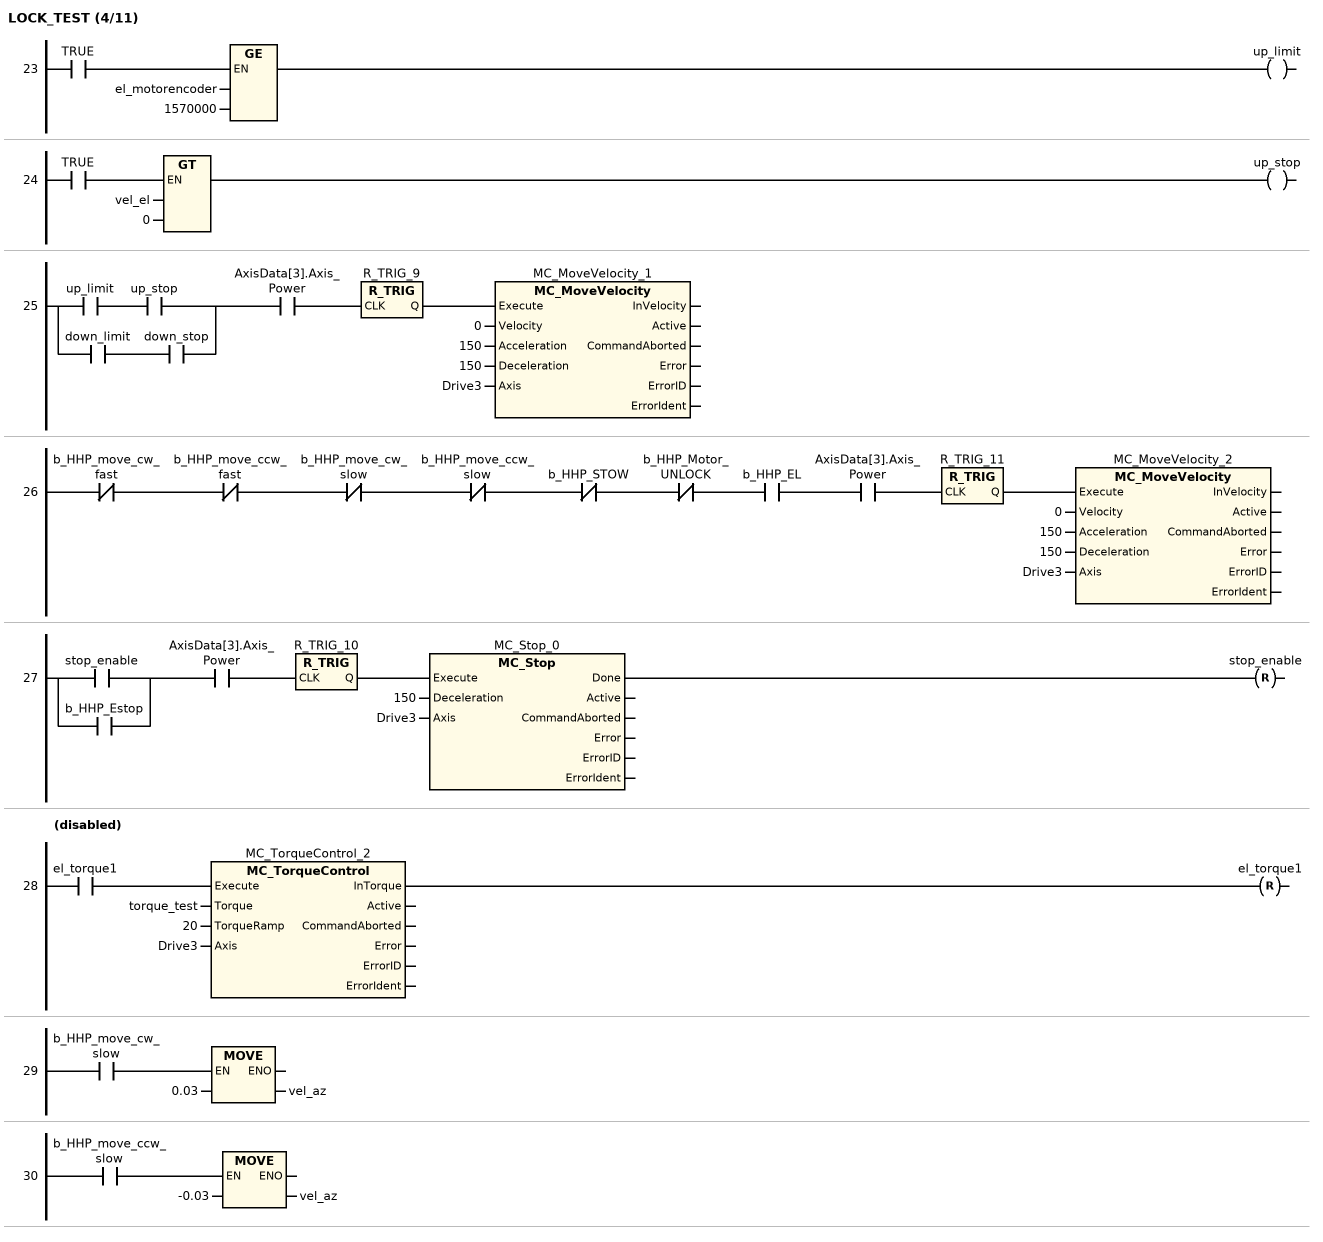
// NETWORK 23
up_limit := el_motorencoder >= 1570000;

// NETWORK 24
up_stop := vel_el > 0;

// NETWORK 25
R_TRIG_9(CLK := (up_limit AND up_stop OR down_limit AND down_stop) AND AxisData[3].Axis_Power); // R_TRIG
MC_MoveVelocity_1(
    Execute := R_TRIG_9.Q,
    Velocity := 0,
    Acceleration := 150,
    Deceleration := 150,
    Axis := Drive3); // MC_MoveVelocity

// NETWORK 26
R_TRIG_11(CLK := NOT b_HHP_move_cw_fast AND NOT b_HHP_move_ccw_fast AND NOT b_HHP_move_cw_slow AND NOT b_HHP_move_ccw_slow AND NOT b_HHP_STOW AND NOT b_HHP_Motor_UNLOCK AND b_HHP_EL AND AxisData[3].Axis_Power); // R_TRIG
MC_MoveVelocity_2(
    Execute := R_TRIG_11.Q,
    Velocity := 0,
    Acceleration := 150,
    Deceleration := 150,
    Axis := Drive3); // MC_MoveVelocity

// NETWORK 27
R_TRIG_10(CLK := (stop_enable OR b_HHP_Estop) AND AxisData[3].Axis_Power); // R_TRIG
MC_Stop_0(Execute := R_TRIG_10.Q, Deceleration := 150, Axis := Drive3); // MC_Stop
stop_enable R= MC_Stop_0.Done;

// NETWORK 28 (disabled)
// MC_TorqueControl_2(Execute := el_torque1, Torque := torque_test, TorqueRamp := 20, Axis := Drive3); // MC_TorqueControl
// el_torque1 R= MC_TorqueControl_2.InTorque;

// NETWORK 29
IF b_HHP_move_cw_slow THEN vel_az := 0.03; END_IF

// NETWORK 30
IF b_HHP_move_ccw_slow THEN vel_az := -0.03; END_IF

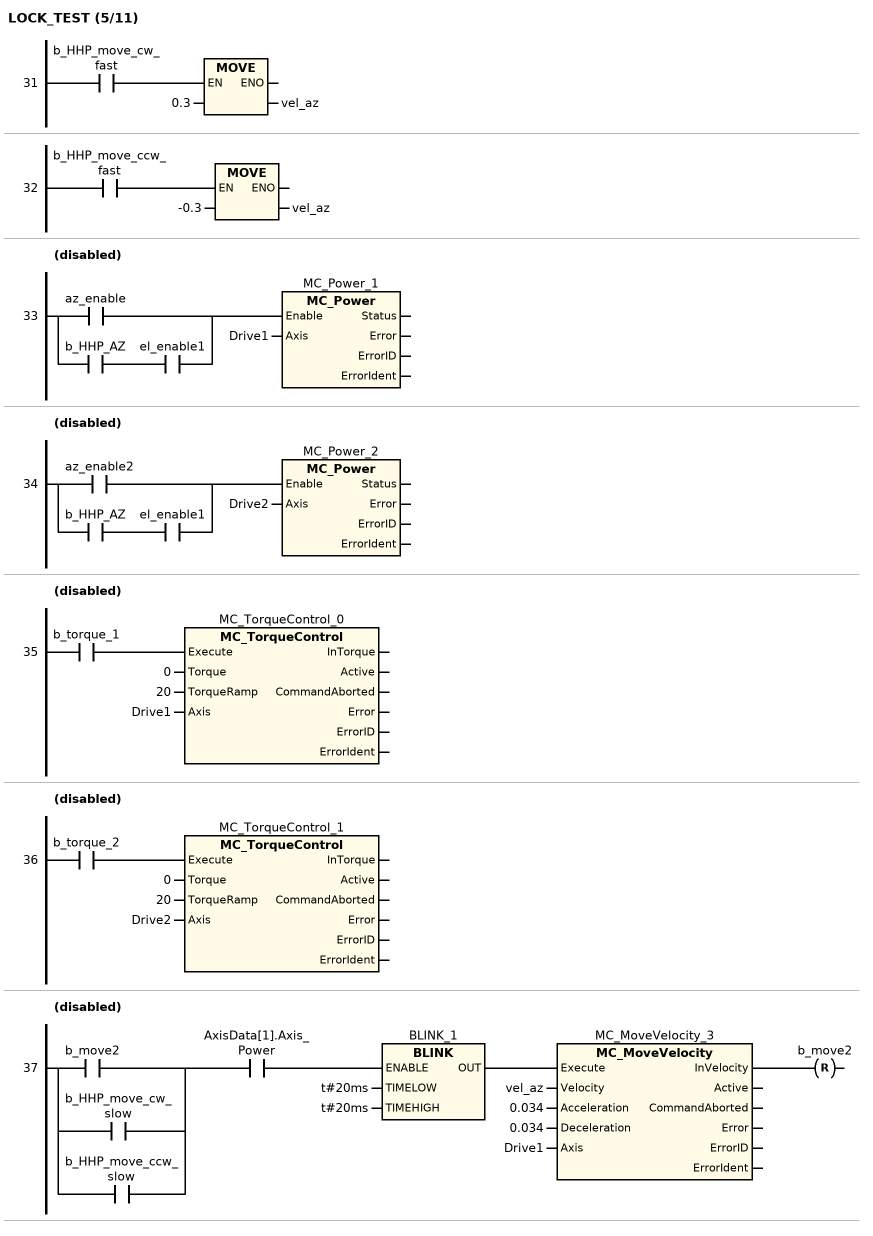
// NETWORK 31
IF b_HHP_move_cw_fast THEN vel_az := 0.3; END_IF

// NETWORK 32
IF b_HHP_move_ccw_fast THEN vel_az := -0.3; END_IF

// NETWORK 33 (disabled)
// MC_Power_1(Enable := az_enable OR b_HHP_AZ AND el_enable1, Axis := Drive1); // MC_Power

// NETWORK 34 (disabled)
// MC_Power_2(Enable := az_enable2 OR b_HHP_AZ AND el_enable1, Axis := Drive2); // MC_Power

// NETWORK 35 (disabled)
// MC_TorqueControl_0(Execute := b_torque_1, Torque := 0, TorqueRamp := 20, Axis := Drive1); // MC_TorqueControl

// NETWORK 36 (disabled)
// MC_TorqueControl_1(Execute := b_torque_2, Torque := 0, TorqueRamp := 20, Axis := Drive2); // MC_TorqueControl

// NETWORK 37 (disabled)
// BLINK_1(
//     ENABLE := (b_move2 OR b_HHP_move_cw_slow OR b_HHP_move_ccw_slow) AND AxisData[1].Axis_Power,
//     TIMELOW := t#20ms,
//     TIMEHIGH := t#20ms); // BLINK
// MC_MoveVelocity_3(
//     Execute := BLINK_1.OUT,
//     Velocity := vel_az,
//     Acceleration := 0.034,
//     Deceleration := 0.034,
//     Axis := Drive1); // MC_MoveVelocity
// b_move2 R= MC_MoveVelocity_3.InVelocity;

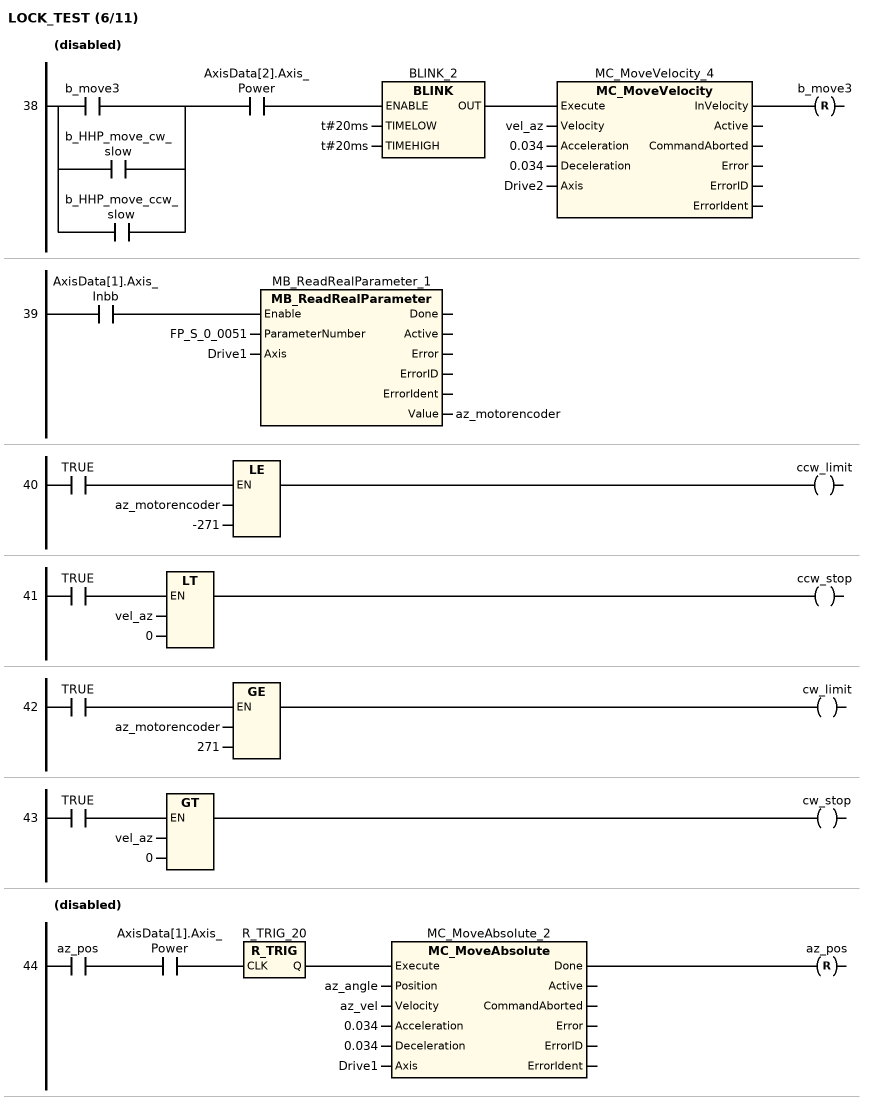
// NETWORK 38 (disabled)
// BLINK_2(
//     ENABLE := (b_move3 OR b_HHP_move_cw_slow OR b_HHP_move_ccw_slow) AND AxisData[2].Axis_Power,
//     TIMELOW := t#20ms,
//     TIMEHIGH := t#20ms); // BLINK
// MC_MoveVelocity_4(
//     Execute := BLINK_2.OUT,
//     Velocity := vel_az,
//     Acceleration := 0.034,
//     Deceleration := 0.034,
//     Axis := Drive2); // MC_MoveVelocity
// b_move3 R= MC_MoveVelocity_4.InVelocity;

// NETWORK 39
MB_ReadRealParameter_1(
    Enable := AxisData[1].Axis_Inbb,
    ParameterNumber := FP_S_0_0051,
    Axis := Drive1,
    Value => az_motorencoder); // MB_ReadRealParameter

// NETWORK 40
ccw_limit := az_motorencoder <= -271;

// NETWORK 41
ccw_stop := vel_az < 0;

// NETWORK 42
cw_limit := az_motorencoder >= 271;

// NETWORK 43
cw_stop := vel_az > 0;

// NETWORK 44 (disabled)
// R_TRIG_20(CLK := az_pos AND AxisData[1].Axis_Power); // R_TRIG
// MC_MoveAbsolute_2(
//     Execute := R_TRIG_20.Q,
//     Position := az_angle,
//     Velocity := az_vel,
//     Acceleration := 0.034,
//     Deceleration := 0.034,
//     Axis := Drive1); // MC_MoveAbsolute
// az_pos R= MC_MoveAbsolute_2.Done;

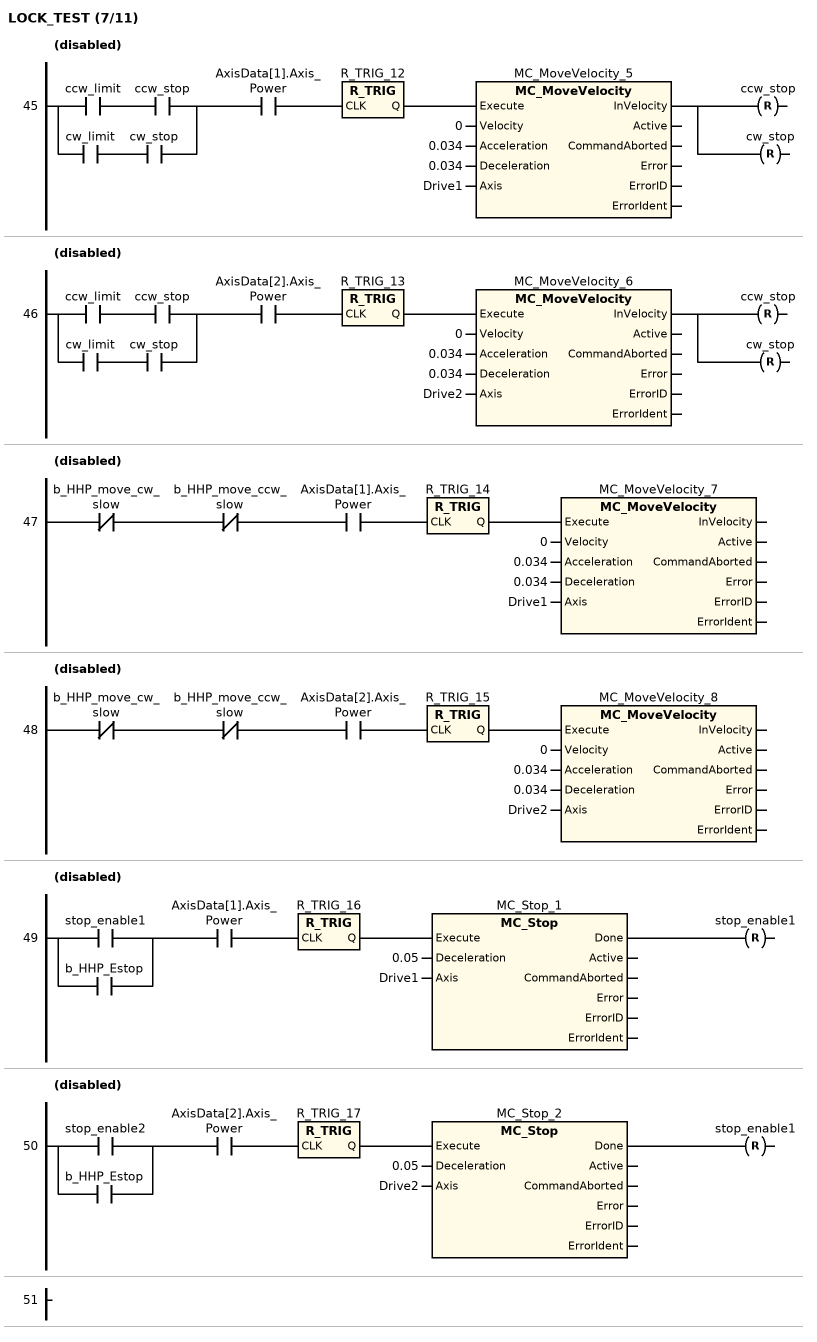
// NETWORK 45 (disabled)
// R_TRIG_12(CLK := (ccw_limit AND ccw_stop OR cw_limit AND cw_stop) AND AxisData[1].Axis_Power); // R_TRIG
// MC_MoveVelocity_5(
//     Execute := R_TRIG_12.Q,
//     Velocity := 0,
//     Acceleration := 0.034,
//     Deceleration := 0.034,
//     Axis := Drive1); // MC_MoveVelocity
// ccw_stop R= MC_MoveVelocity_5.InVelocity;
// cw_stop R= MC_MoveVelocity_5.InVelocity;

// NETWORK 46 (disabled)
// R_TRIG_13(CLK := (ccw_limit AND ccw_stop OR cw_limit AND cw_stop) AND AxisData[2].Axis_Power); // R_TRIG
// MC_MoveVelocity_6(
//     Execute := R_TRIG_13.Q,
//     Velocity := 0,
//     Acceleration := 0.034,
//     Deceleration := 0.034,
//     Axis := Drive2); // MC_MoveVelocity
// ccw_stop R= MC_MoveVelocity_6.InVelocity;
// cw_stop R= MC_MoveVelocity_6.InVelocity;

// NETWORK 47 (disabled)
// R_TRIG_14(CLK := NOT b_HHP_move_cw_slow AND NOT b_HHP_move_ccw_slow AND AxisData[1].Axis_Power); // R_TRIG
// MC_MoveVelocity_7(
//     Execute := R_TRIG_14.Q,
//     Velocity := 0,
//     Acceleration := 0.034,
//     Deceleration := 0.034,
//     Axis := Drive1); // MC_MoveVelocity

// NETWORK 48 (disabled)
// R_TRIG_15(CLK := NOT b_HHP_move_cw_slow AND NOT b_HHP_move_ccw_slow AND AxisData[2].Axis_Power); // R_TRIG
// MC_MoveVelocity_8(
//     Execute := R_TRIG_15.Q,
//     Velocity := 0,
//     Acceleration := 0.034,
//     Deceleration := 0.034,
//     Axis := Drive2); // MC_MoveVelocity

// NETWORK 49 (disabled)
// R_TRIG_16(CLK := (stop_enable1 OR b_HHP_Estop) AND AxisData[1].Axis_Power); // R_TRIG
// MC_Stop_1(Execute := R_TRIG_16.Q, Deceleration := 0.05, Axis := Drive1); // MC_Stop
// stop_enable1 R= MC_Stop_1.Done;

// NETWORK 50 (disabled)
// R_TRIG_17(CLK := (stop_enable2 OR b_HHP_Estop) AND AxisData[2].Axis_Power); // R_TRIG
// MC_Stop_2(Execute := R_TRIG_17.Q, Deceleration := 0.05, Axis := Drive2); // MC_Stop
// stop_enable1 R= MC_Stop_2.Done;

// NETWORK 51

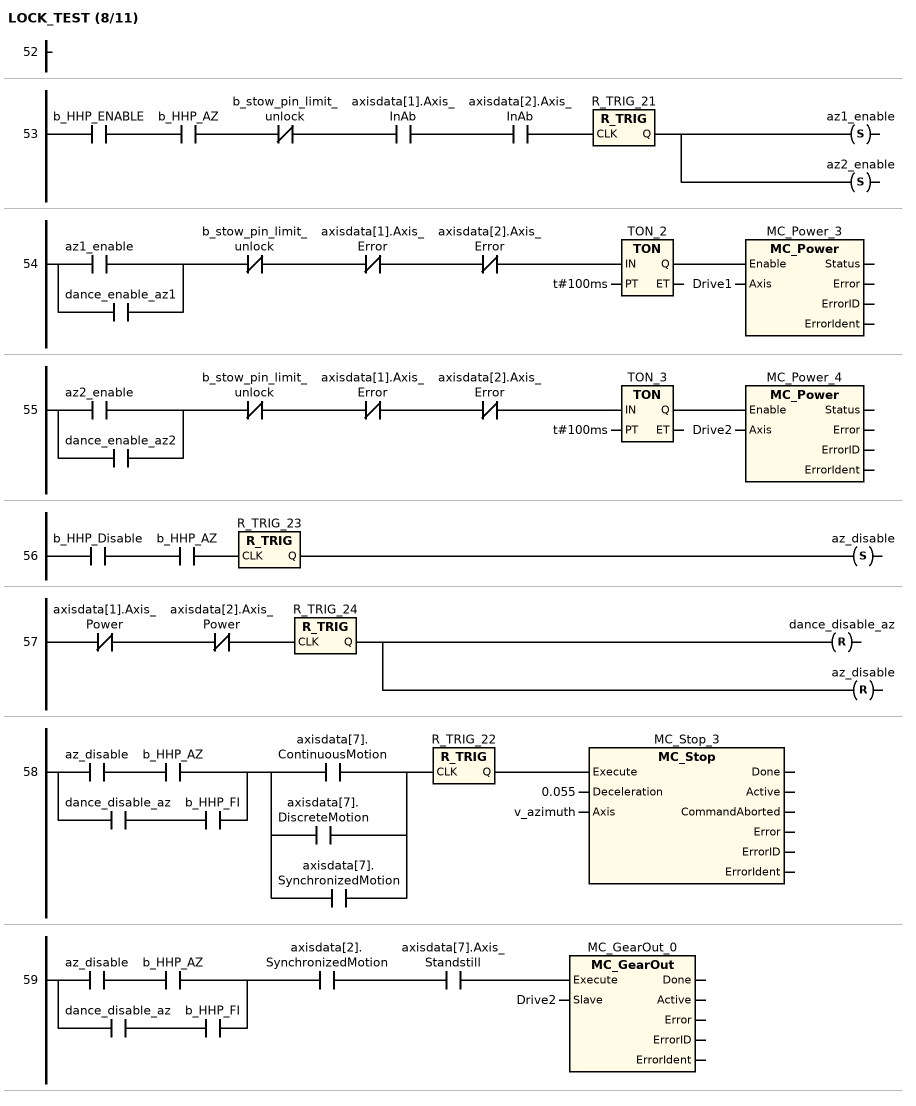
// NETWORK 52

// NETWORK 53
R_TRIG_21(CLK := b_HHP_ENABLE AND b_HHP_AZ AND NOT b_stow_pin_limit_unlock AND axisdata[1].Axis_InAb AND axisdata[2].Axis_InAb); // R_TRIG
az1_enable S= R_TRIG_21.Q;
az2_enable S= R_TRIG_21.Q;

// NETWORK 54
TON_2(IN := (az1_enable OR dance_enable_az1) AND NOT b_stow_pin_limit_unlock AND NOT axisdata[1].Axis_Error AND NOT axisdata[2].Axis_Error, PT := t#100ms); // TON
MC_Power_3(Enable := TON_2.Q, Axis := Drive1); // MC_Power

// NETWORK 55
TON_3(IN := (az2_enable OR dance_enable_az2) AND NOT b_stow_pin_limit_unlock AND NOT axisdata[1].Axis_Error AND NOT axisdata[2].Axis_Error, PT := t#100ms); // TON
MC_Power_4(Enable := TON_3.Q, Axis := Drive2); // MC_Power

// NETWORK 56
R_TRIG_23(CLK := b_HHP_Disable AND b_HHP_AZ); // R_TRIG
az_disable S= R_TRIG_23.Q;

// NETWORK 57
R_TRIG_24(CLK := NOT axisdata[1].Axis_Power AND NOT axisdata[2].Axis_Power); // R_TRIG
dance_disable_az R= R_TRIG_24.Q;
az_disable R= R_TRIG_24.Q;

// NETWORK 58
R_TRIG_22(CLK := (az_disable AND b_HHP_AZ OR dance_disable_az AND b_HHP_FI) AND (axisdata[7].ContinuousMotion OR axisdata[7].DiscreteMotion OR axisdata[7].SynchronizedMotion)); // R_TRIG
MC_Stop_3(Execute := R_TRIG_22.Q, Deceleration := 0.055, Axis := v_azimuth); // MC_Stop

// NETWORK 59
MC_GearOut_0(Execute := (az_disable AND b_HHP_AZ OR dance_disable_az AND b_HHP_FI) AND axisdata[2].SynchronizedMotion AND axisdata[7].Axis_Standstill, Slave := Drive2); // MC_GearOut

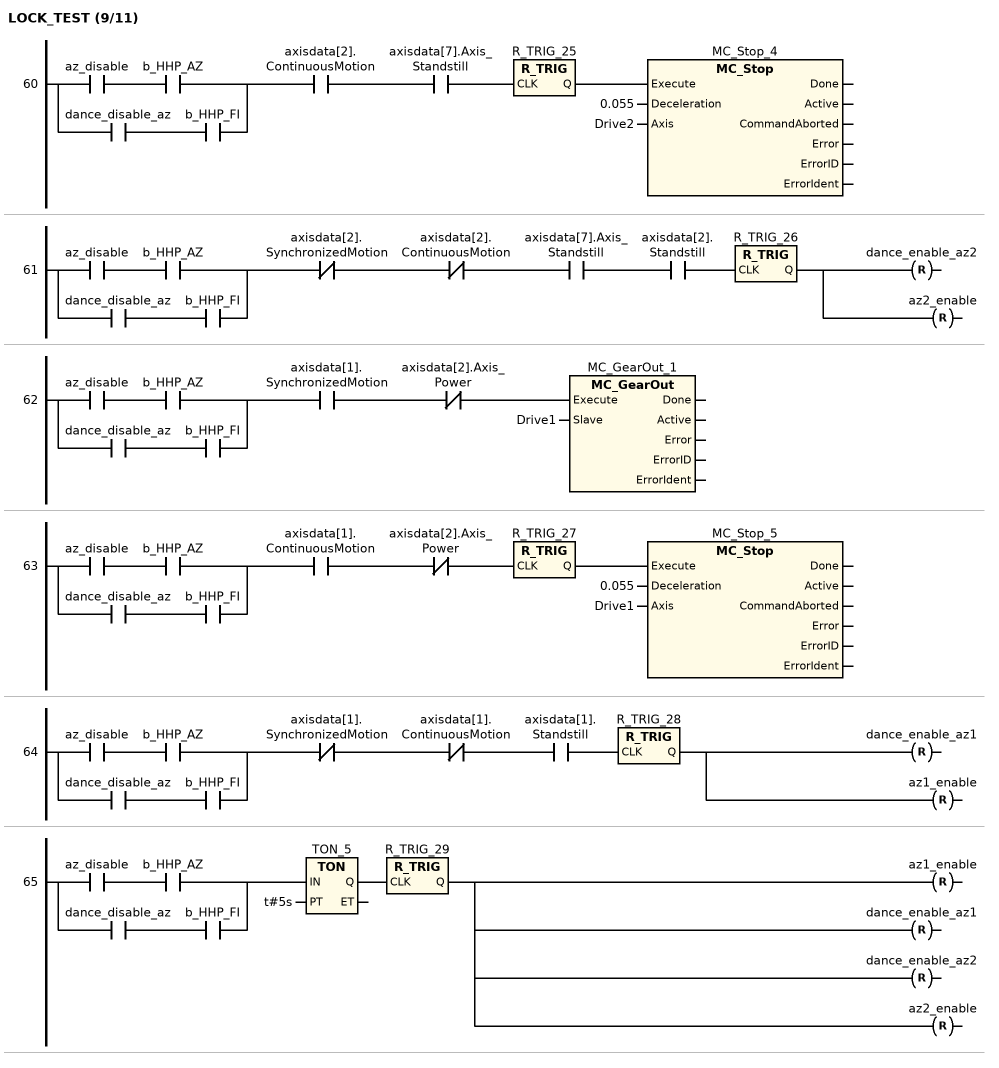
// NETWORK 60
R_TRIG_25(CLK := (az_disable AND b_HHP_AZ OR dance_disable_az AND b_HHP_FI) AND axisdata[2].ContinuousMotion AND axisdata[7].Axis_Standstill); // R_TRIG
MC_Stop_4(Execute := R_TRIG_25.Q, Deceleration := 0.055, Axis := Drive2); // MC_Stop

// NETWORK 61
R_TRIG_26(CLK := (az_disable AND b_HHP_AZ OR dance_disable_az AND b_HHP_FI) AND NOT axisdata[2].SynchronizedMotion AND NOT axisdata[2].ContinuousMotion AND axisdata[7].Axis_Standstill AND axisdata[2].Standstill); // R_TRIG
dance_enable_az2 R= R_TRIG_26.Q;
az2_enable R= R_TRIG_26.Q;

// NETWORK 62
MC_GearOut_1(Execute := (az_disable AND b_HHP_AZ OR dance_disable_az AND b_HHP_FI) AND axisdata[1].SynchronizedMotion AND NOT axisdata[2].Axis_Power, Slave := Drive1); // MC_GearOut

// NETWORK 63
R_TRIG_27(CLK := (az_disable AND b_HHP_AZ OR dance_disable_az AND b_HHP_FI) AND axisdata[1].ContinuousMotion AND NOT axisdata[2].Axis_Power); // R_TRIG
MC_Stop_5(Execute := R_TRIG_27.Q, Deceleration := 0.055, Axis := Drive1); // MC_Stop

// NETWORK 64
R_TRIG_28(CLK := (az_disable AND b_HHP_AZ OR dance_disable_az AND b_HHP_FI) AND NOT axisdata[1].SynchronizedMotion AND NOT axisdata[1].ContinuousMotion AND axisdata[1].Standstill); // R_TRIG
dance_enable_az1 R= R_TRIG_28.Q;
az1_enable R= R_TRIG_28.Q;

// NETWORK 65
TON_5(IN := az_disable AND b_HHP_AZ OR dance_disable_az AND b_HHP_FI, PT := t#5s); // TON
R_TRIG_29(CLK := TON_5.Q); // R_TRIG
az1_enable R= R_TRIG_29.Q;
dance_enable_az1 R= R_TRIG_29.Q;
dance_enable_az2 R= R_TRIG_29.Q;
az2_enable R= R_TRIG_29.Q;

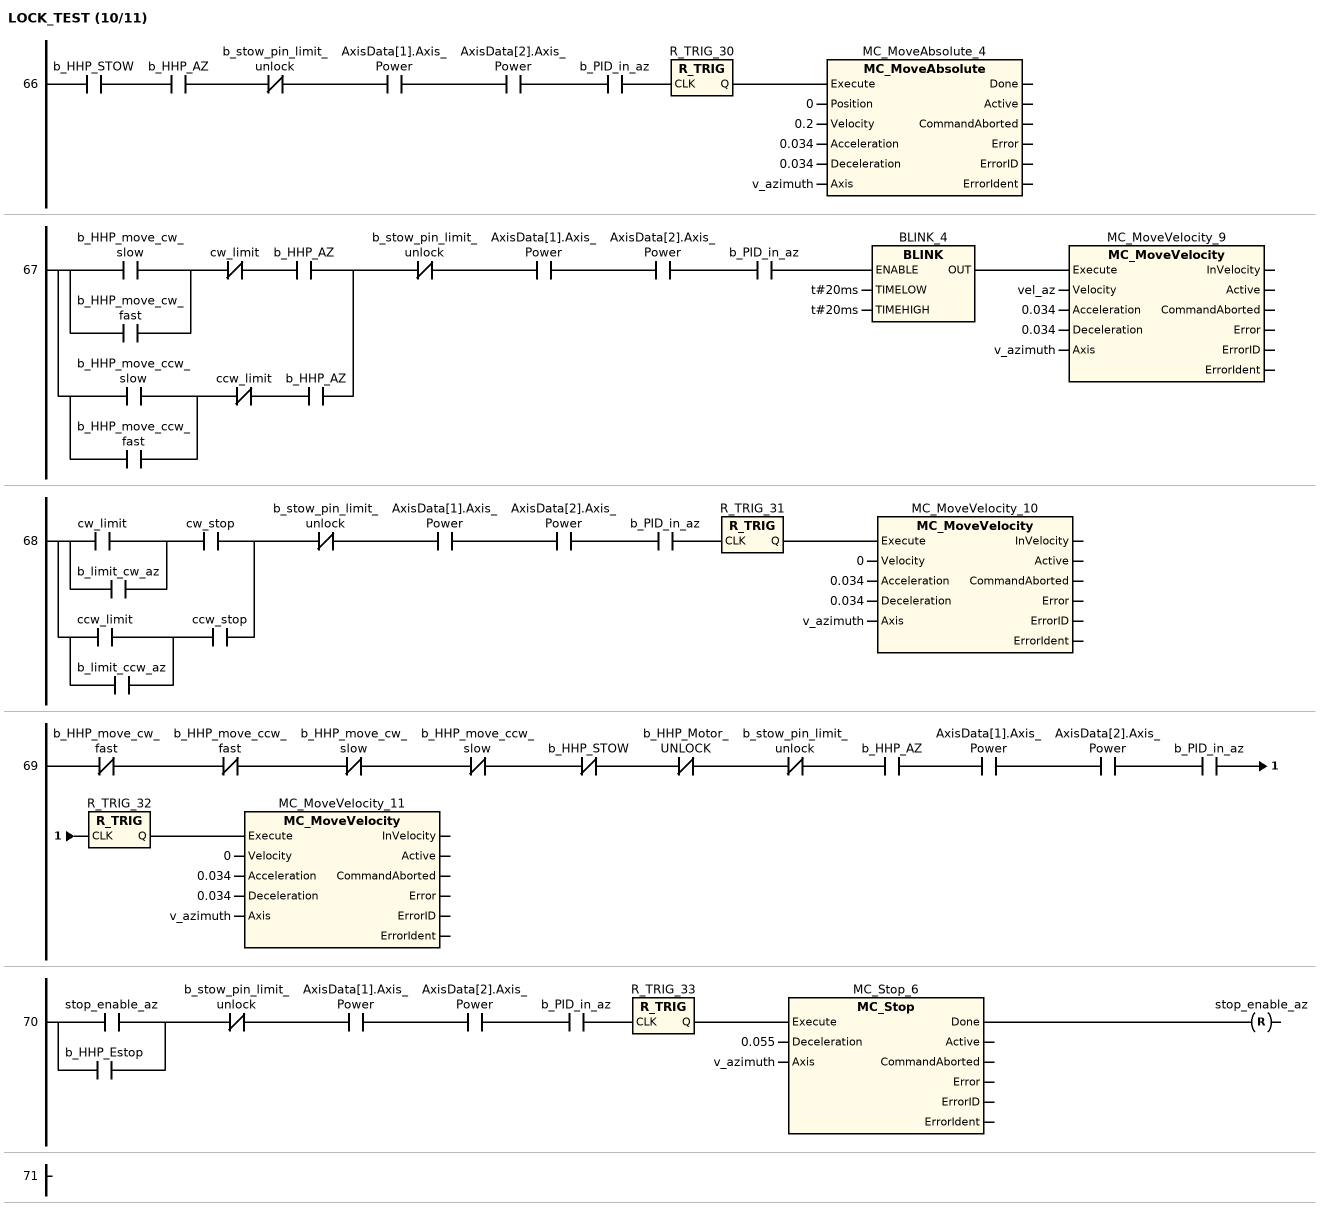
// NETWORK 66
R_TRIG_30(CLK := b_HHP_STOW AND b_HHP_AZ AND NOT b_stow_pin_limit_unlock AND AxisData[1].Axis_Power AND AxisData[2].Axis_Power AND b_PID_in_az); // R_TRIG
MC_MoveAbsolute_4(
    Execute := R_TRIG_30.Q,
    Position := 0,
    Velocity := 0.2,
    Acceleration := 0.034,
    Deceleration := 0.034,
    Axis := v_azimuth); // MC_MoveAbsolute

// NETWORK 67
BLINK_4(
    ENABLE := ((b_HHP_move_cw_slow OR b_HHP_move_cw_fast) AND NOT cw_limit AND b_HHP_AZ OR (b_HHP_move_ccw_slow OR b_HHP_move_ccw_fast) AND NOT ccw_limit AND b_HHP_AZ) AND NOT b_stow_pin_limit_unlock AND AxisData[1].Axis_Power AND AxisData[2].Axis_Power AND b_PID_in_az,
    TIMELOW := t#20ms,
    TIMEHIGH := t#20ms); // BLINK
MC_MoveVelocity_9(
    Execute := BLINK_4.OUT,
    Velocity := vel_az,
    Acceleration := 0.034,
    Deceleration := 0.034,
    Axis := v_azimuth); // MC_MoveVelocity

// NETWORK 68
R_TRIG_31(CLK := ((cw_limit OR b_limit_cw_az) AND cw_stop OR (ccw_limit OR b_limit_ccw_az) AND ccw_stop) AND NOT b_stow_pin_limit_unlock AND AxisData[1].Axis_Power AND AxisData[2].Axis_Power AND b_PID_in_az); // R_TRIG
MC_MoveVelocity_10(
    Execute := R_TRIG_31.Q,
    Velocity := 0,
    Acceleration := 0.034,
    Deceleration := 0.034,
    Axis := v_azimuth); // MC_MoveVelocity

// NETWORK 69
R_TRIG_32(CLK := NOT b_HHP_move_cw_fast AND NOT b_HHP_move_ccw_fast AND NOT b_HHP_move_cw_slow AND NOT b_HHP_move_ccw_slow AND NOT b_HHP_STOW AND NOT b_HHP_Motor_UNLOCK AND NOT b_stow_pin_limit_unlock AND b_HHP_AZ AND AxisData[1].Axis_Power AND AxisData[2].Axis_Power AND b_PID_in_az); // R_TRIG
MC_MoveVelocity_11(
    Execute := R_TRIG_32.Q,
    Velocity := 0,
    Acceleration := 0.034,
    Deceleration := 0.034,
    Axis := v_azimuth); // MC_MoveVelocity

// NETWORK 70
R_TRIG_33(CLK := (stop_enable_az OR b_HHP_Estop) AND NOT b_stow_pin_limit_unlock AND AxisData[1].Axis_Power AND AxisData[2].Axis_Power AND b_PID_in_az); // R_TRIG
MC_Stop_6(Execute := R_TRIG_33.Q, Deceleration := 0.055, Axis := v_azimuth); // MC_Stop
stop_enable_az R= MC_Stop_6.Done;

// NETWORK 71

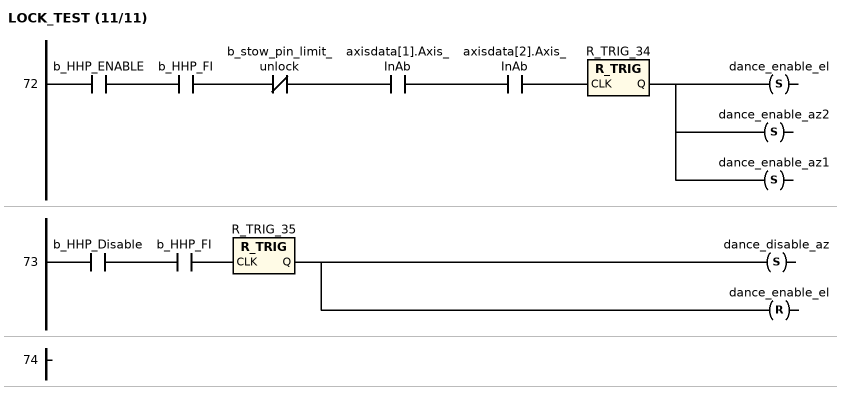
// NETWORK 72
R_TRIG_34(CLK := b_HHP_ENABLE AND b_HHP_FI AND NOT b_stow_pin_limit_unlock AND axisdata[1].Axis_InAb AND axisdata[2].Axis_InAb); // R_TRIG
dance_enable_el S= R_TRIG_34.Q;
dance_enable_az2 S= R_TRIG_34.Q;
dance_enable_az1 S= R_TRIG_34.Q;

// NETWORK 73
R_TRIG_35(CLK := b_HHP_Disable AND b_HHP_FI); // R_TRIG
dance_disable_az S= R_TRIG_35.Q;
dance_enable_el R= R_TRIG_35.Q;

// NETWORK 74

END_PROGRAM

// IndraMotionMlc1/Application/POUs/Motion/P_power_on_Sim
(*the program is built for power on the 3 axis under the contol of remote or local.
the elevation axis is the similar with the azimuth*)
PROGRAM P_power_on_Sim
VAR
(*<<<<<<<<definition of r_trig for detecting a rising edge>>>>>>>>>>>>>>*)
	fb_rtrig_p1: R_TRIG;
	fb_rtrig_p3: R_TRIG;
	fb_rtrig_p5: R_TRIG;
	fb_rtrig_az: R_TRIG;
	fb_rtrig_el: R_TRIG;
	fb_rtrig_FI: R_TRIG;
	fb_rtrig_en_remote: R_TRIG;
	fb_rtrig_en_TCP: R_TRIG;
(*<<<<<<<The function block Timer On Delay implements a turn-on delay>>>>>>*)
	ton_en_1: TON;
	ton_en_2: TON;
	ton_en_3: TON;
	ton_en_4: TON;
	ton_en_5: TON;
	ton_en_6: TON;
(*MC_Power function block controls the power connection (power on or off)*)
	FB_1_power: MC_Power;
	FB_2_power: MC_Power;
	FB_3_power: MC_Power;
	FB_4_power: MC_Power;
	FB_5_power: MC_Power;
	FB_6_power: MC_Power;
	b_1_enable_on: BOOL;
	b_2_enable_on: BOOL;
	b_3_enable_on: BOOL;
	b_4_enable_on: BOOL;
	b_5_enable_on: BOOL;
	b_6_enable_on: BOOL;
(*With "MB_GearInPos",it is possible to realize a motion of the slave axis which is phase synchronous to the master axis*)
	fb_gearinPos_1: MB_GearInPos;
	fb_gearin_2: MB_GearInPos;
	fb_gearinPos_3: MB_GearInPos;
	fb_gearin_4: MB_GearInPos;
	fb_gearinPos_5: MB_GearInPos;
	fb_gearin_6: MB_GearInPos;
	b_gearin_1_done: BOOL;
	
	b_gearin_5_done:BOOL;
(*"MC_MoveAbsolute" is used to move the drive to a preset absolute position.*)
	FB_move_master_az: MC_MoveAbsolute;
	FB_move_master_el: MC_MoveAbsolute;
	FB_move_master_FI: MC_MoveAbsolute;
	b_M_az_done: BOOL;
	b_M_el_done: BOOL;
	b_M_FI_done: BOOL;
(*MB_Home function block controls axes with incremental encoder when executing the "search home" sequence*)
	fb_home_az2: MB_Home;
	fb_home_el2: MB_Home;
	fb_home_FI2: MB_Home;
	b_home_az2_done: BOOL;
	b_home_el2_done: BOOL;
	b_home_FI2_done: BOOL;
(*<<<<<<<<<<<<<<<<<<<<<<<<<<<<<clear error>>>>>>>>>>>>>>>>>>>>>>>>>>>>>>>>>*)
	TCP_clear_error: BOOL;
	FB_clear_error_TCP: MB_WriteParameter;
	TCP_clear_done: BOOL;
(*add 2011 06 09 to delete 1sec delay*)
	fb_gearinPos_el: MB_GearInPos;
	b_gearin_el_done: BOOL;
	fb_gearout_el: MC_GearOut;
	rtrig_set_gearin_3: R_TRIG;
	b_gearin_3: BOOL;
	rtrig_reset_gearin_3: F_TRIG;
	ton_clear_on: TON;
	fb_gearinPos_FI: MB_GearInPos;
	test_111: BOOL;
	ssss: BOOL;
	test1: BOOL;
	test2: BOOL;
	test3: BOOL;
	TON_enable_az: ton;
	TON_enable_az2: ton;
	fb_gearPos_2: MB_GearInPos;
	TON_enable_el: ton;
	b_M_el_done_1: BOOL;
	R_TRIG_0: R_TRIG;
END_VAR

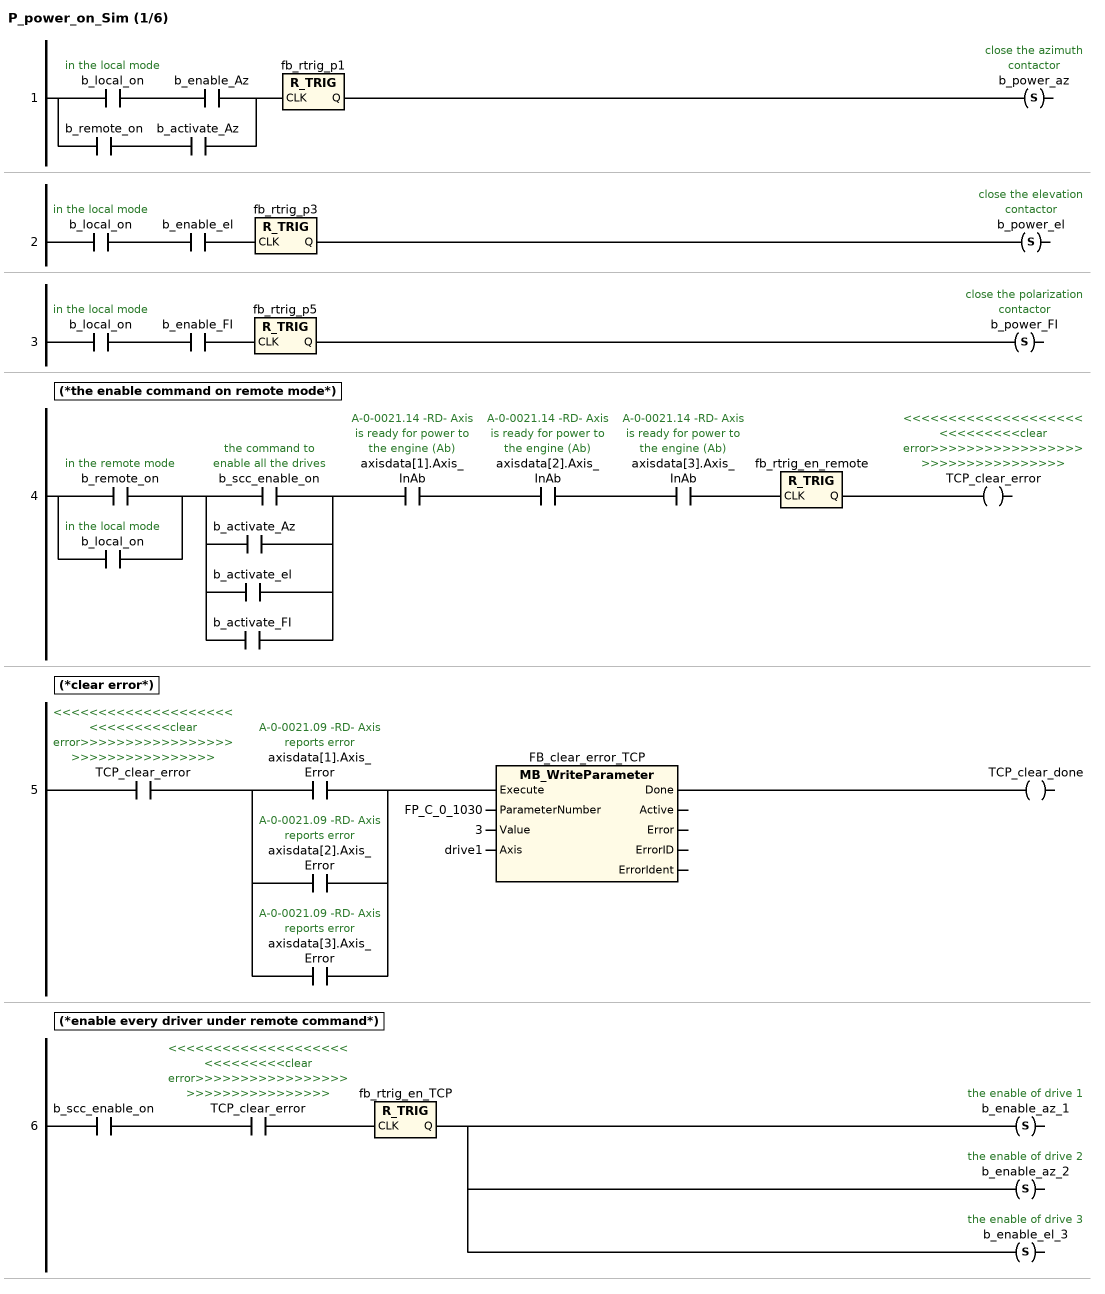
// NETWORK 1
//   fb_rtrig_p1: <<<<<<<<definition of r_trig for detecting a rising edge>>>>>>>>>>>>>>
//   b_local_on: in the local mode
//   b_power_az: close the azimuth contactor
fb_rtrig_p1(CLK := b_local_on AND b_enable_Az OR b_remote_on AND b_activate_Az); // R_TRIG
b_power_az S= fb_rtrig_p1.Q;

// NETWORK 2
//   b_local_on: in the local mode
//   b_power_el: close the elevation contactor
fb_rtrig_p3(CLK := b_local_on AND b_enable_el); // R_TRIG
b_power_el S= fb_rtrig_p3.Q;

// NETWORK 3
//   b_local_on: in the local mode
//   b_power_FI: close the polarization contactor
fb_rtrig_p5(CLK := b_local_on AND b_enable_FI); // R_TRIG
b_power_FI S= fb_rtrig_p5.Q;

// NETWORK 4
//   b_remote_on: in the remote mode
//   b_local_on: in the local mode
//   b_scc_enable_on: the command to enable all the drives
//   axisdata[1].Axis_InAb: A-0-0021.14 -RD- Axis is ready for power to the engine (Ab)
//   axisdata[2].Axis_InAb: A-0-0021.14 -RD- Axis is ready for power to the engine (Ab)
//   axisdata[3].Axis_InAb: A-0-0021.14 -RD- Axis is ready for power to the engine (Ab)
//   TCP_clear_error: <<<<<<<<<<<<<<<<<<<<<<<<<<<<<clear error>>>>>>>>>>>>>>>>>>>>>>>>>>>>>>>>>
// label: (*the enable command on remote mode*)
fb_rtrig_en_remote(CLK := (b_remote_on OR b_local_on) AND (b_scc_enable_on OR b_activate_Az OR b_activate_el OR b_activate_FI) AND axisdata[1].Axis_InAb AND axisdata[2].Axis_InAb AND axisdata[3].Axis_InAb); // R_TRIG
TCP_clear_error := fb_rtrig_en_remote.Q;

// NETWORK 5
//   TCP_clear_error: <<<<<<<<<<<<<<<<<<<<<<<<<<<<<clear error>>>>>>>>>>>>>>>>>>>>>>>>>>>>>>>>>
//   axisdata[1].Axis_Error: A-0-0021.09 -RD- Axis reports error
//   axisdata[2].Axis_Error: A-0-0021.09 -RD- Axis reports error
//   axisdata[3].Axis_Error: A-0-0021.09 -RD- Axis reports error
//   FP_C_0_1030: Command: Clear all control errors
//   drive1: Real axis "Drive1" with axis number 1
// label: (*clear error*)
FB_clear_error_TCP(
    Execute := TCP_clear_error AND (axisdata[1].Axis_Error OR axisdata[2].Axis_Error OR axisdata[3].Axis_Error),
    ParameterNumber := FP_C_0_1030,
    Value := 3,
    Axis := drive1); // MB_WriteParameter
TCP_clear_done := FB_clear_error_TCP.Done;

// NETWORK 6
//   TCP_clear_error: <<<<<<<<<<<<<<<<<<<<<<<<<<<<<clear error>>>>>>>>>>>>>>>>>>>>>>>>>>>>>>>>>
//   b_enable_az_1: the enable of drive 1
//   b_enable_az_2: the enable of drive 2
//   b_enable_el_3: the enable of drive 3
// label: (*enable every driver under remote command*)
fb_rtrig_en_TCP(CLK := b_scc_enable_on AND TCP_clear_error); // R_TRIG
b_enable_az_1 S= fb_rtrig_en_TCP.Q;
b_enable_az_2 S= fb_rtrig_en_TCP.Q;
b_enable_el_3 S= fb_rtrig_en_TCP.Q;

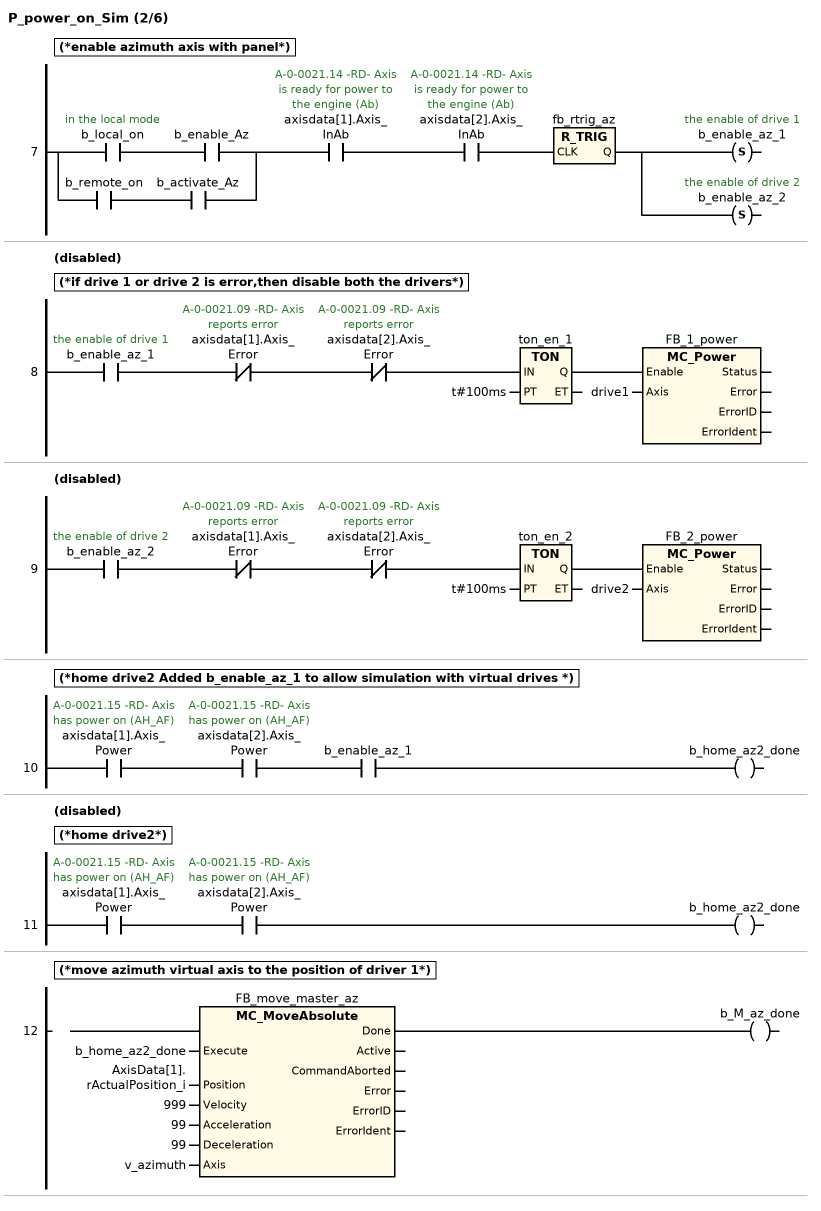
// NETWORK 7
//   b_local_on: in the local mode
//   axisdata[1].Axis_InAb: A-0-0021.14 -RD- Axis is ready for power to the engine (Ab)
//   axisdata[2].Axis_InAb: A-0-0021.14 -RD- Axis is ready for power to the engine (Ab)
//   b_enable_az_1: the enable of drive 1
//   b_enable_az_2: the enable of drive 2
// label: (*enable azimuth axis with panel*)
fb_rtrig_az(CLK := (b_local_on AND b_enable_Az OR b_remote_on AND b_activate_Az) AND axisdata[1].Axis_InAb AND axisdata[2].Axis_InAb); // R_TRIG
b_enable_az_1 S= fb_rtrig_az.Q;
b_enable_az_2 S= fb_rtrig_az.Q;

// NETWORK 8 (disabled)
//   FB_1_power: MC_Power function block controls the power connection (power on or off)
//   ton_en_1: <<<<<<<The function block Timer On Delay implements a turn-on delay>>>>>>
//   b_enable_az_1: the enable of drive 1
//   axisdata[1].Axis_Error: A-0-0021.09 -RD- Axis reports error
//   axisdata[2].Axis_Error: A-0-0021.09 -RD- Axis reports error
//   drive1: Real axis "Drive1" with axis number 1
// label: (*if drive 1 or drive 2 is error,then disable both the drivers*)
// ton_en_1(IN := b_enable_az_1 AND NOT axisdata[1].Axis_Error AND NOT axisdata[2].Axis_Error, PT := t#100ms); // TON
// FB_1_power(Enable := ton_en_1.Q, Axis := drive1); // MC_Power

// NETWORK 9 (disabled)
//   b_enable_az_2: the enable of drive 2
//   axisdata[1].Axis_Error: A-0-0021.09 -RD- Axis reports error
//   axisdata[2].Axis_Error: A-0-0021.09 -RD- Axis reports error
//   drive2: Real axis "Drive2" with axis number 2
// ton_en_2(IN := b_enable_az_2 AND NOT axisdata[1].Axis_Error AND NOT axisdata[2].Axis_Error, PT := t#100ms); // TON
// FB_2_power(Enable := ton_en_2.Q, Axis := drive2); // MC_Power

// NETWORK 10
//   axisdata[1].Axis_Power: A-0-0021.15 -RD- Axis has power on (AH_AF)
//   axisdata[2].Axis_Power: A-0-0021.15 -RD- Axis has power on (AH_AF)
// label: (*home drive2 Added b_enable_az_1 to allow simulation with virtual drives *)
b_home_az2_done := axisdata[1].Axis_Power AND axisdata[2].Axis_Power AND b_enable_az_1;

// NETWORK 11 (disabled)
//   axisdata[1].Axis_Power: A-0-0021.15 -RD- Axis has power on (AH_AF)
//   axisdata[2].Axis_Power: A-0-0021.15 -RD- Axis has power on (AH_AF)
// label: (*home drive2*)
// b_home_az2_done := axisdata[1].Axis_Power AND axisdata[2].Axis_Power;

// NETWORK 12
//   FB_move_master_az: "MC_MoveAbsolute" is used to move the drive to a preset absolute position.
//   AxisData[1].rActualPosition_i: A-0-0100 -RD- Actual position
//   v_azimuth: Virtual axis "v_azimuth" with axis number 7
// label: (*move azimuth virtual axis to the position of driver 1*)
FB_move_master_az(
    Execute := b_home_az2_done,
    Position := AxisData[1].rActualPosition_i,
    Velocity := 999,
    Acceleration := 99,
    Deceleration := 99,
    Axis := v_azimuth); // MC_MoveAbsolute
b_M_az_done := FB_move_master_az.Done;

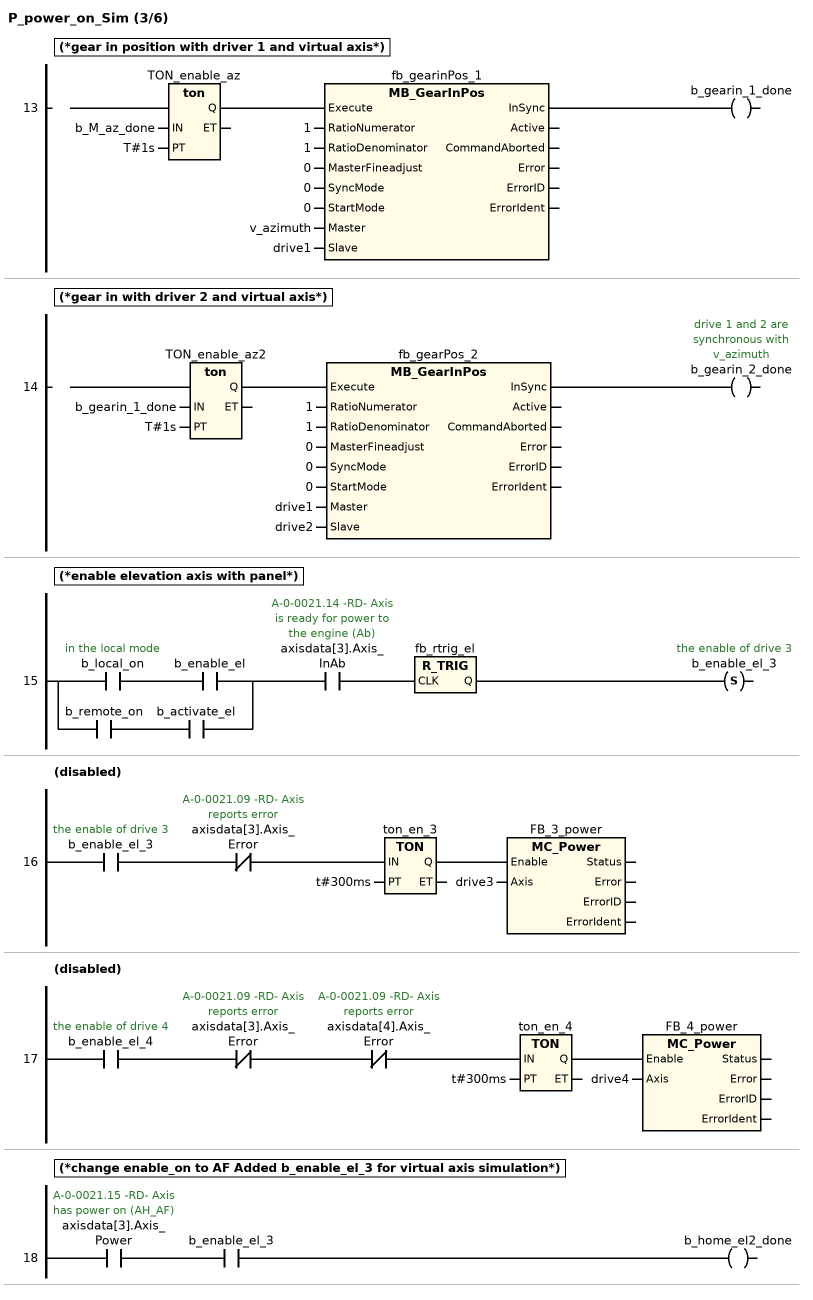
// NETWORK 13
//   fb_gearinPos_1: With "MB_GearInPos",it is possible to realize a motion of the slave axis which is phase synchronous to the master axis
//   v_azimuth: Virtual axis "v_azimuth" with axis number 7
//   drive1: Real axis "Drive1" with axis number 1
// label: (*gear in position with driver 1 and virtual axis*)
TON_enable_az(IN := b_M_az_done, PT := T#1s); // ton
fb_gearinPos_1(
    Execute := TON_enable_az.Q,
    RatioNumerator := 1,
    RatioDenominator := 1,
    MasterFineadjust := 0,
    SyncMode := 0,
    StartMode := 0,
    Master := v_azimuth,
    Slave := drive1); // MB_GearInPos
b_gearin_1_done := fb_gearinPos_1.InSync;

// NETWORK 14
//   drive1: Virtual axis "v_azimuth" with axis number 7
//   drive2: Real axis "Drive2" with axis number 2
//   b_gearin_2_done: drive 1 and 2 are synchronous with v_azimuth
// label: (*gear in with driver 2 and virtual axis*)
TON_enable_az2(IN := b_gearin_1_done, PT := T#1s); // ton
fb_gearPos_2(
    Execute := TON_enable_az2.Q,
    RatioNumerator := 1,
    RatioDenominator := 1,
    MasterFineadjust := 0,
    SyncMode := 0,
    StartMode := 0,
    Master := drive1,
    Slave := drive2); // MB_GearInPos
b_gearin_2_done := fb_gearPos_2.InSync;

// NETWORK 15
//   b_local_on: in the local mode
//   axisdata[3].Axis_InAb: A-0-0021.14 -RD- Axis is ready for power to the engine (Ab)
//   b_enable_el_3: the enable of drive 3
// label: (*enable elevation axis with panel*)
fb_rtrig_el(CLK := (b_local_on AND b_enable_el OR b_remote_on AND b_activate_el) AND axisdata[3].Axis_InAb); // R_TRIG
b_enable_el_3 S= fb_rtrig_el.Q;

// NETWORK 16 (disabled)
//   b_enable_el_3: the enable of drive 3
//   axisdata[3].Axis_Error: A-0-0021.09 -RD- Axis reports error
//   drive3: Real axis "Drive3" with axis number 3
// ton_en_3(IN := b_enable_el_3 AND NOT axisdata[3].Axis_Error, PT := t#300ms); // TON
// FB_3_power(Enable := ton_en_3.Q, Axis := drive3); // MC_Power

// NETWORK 17 (disabled)
//   b_enable_el_4: the enable of drive 4
//   axisdata[3].Axis_Error: A-0-0021.09 -RD- Axis reports error
//   axisdata[4].Axis_Error: A-0-0021.09 -RD- Axis reports error
//   drive4: Real axis "Drive4" with axis number 4
// ton_en_4(IN := b_enable_el_4 AND NOT axisdata[3].Axis_Error AND NOT axisdata[4].Axis_Error, PT := t#300ms); // TON
// FB_4_power(Enable := ton_en_4.Q, Axis := drive4); // MC_Power

// NETWORK 18
//   axisdata[3].Axis_Power: A-0-0021.15 -RD- Axis has power on (AH_AF)
// label: (*change enable_on to AF Added b_enable_el_3 for virtual axis simulation*)
b_home_el2_done := axisdata[3].Axis_Power AND b_enable_el_3;

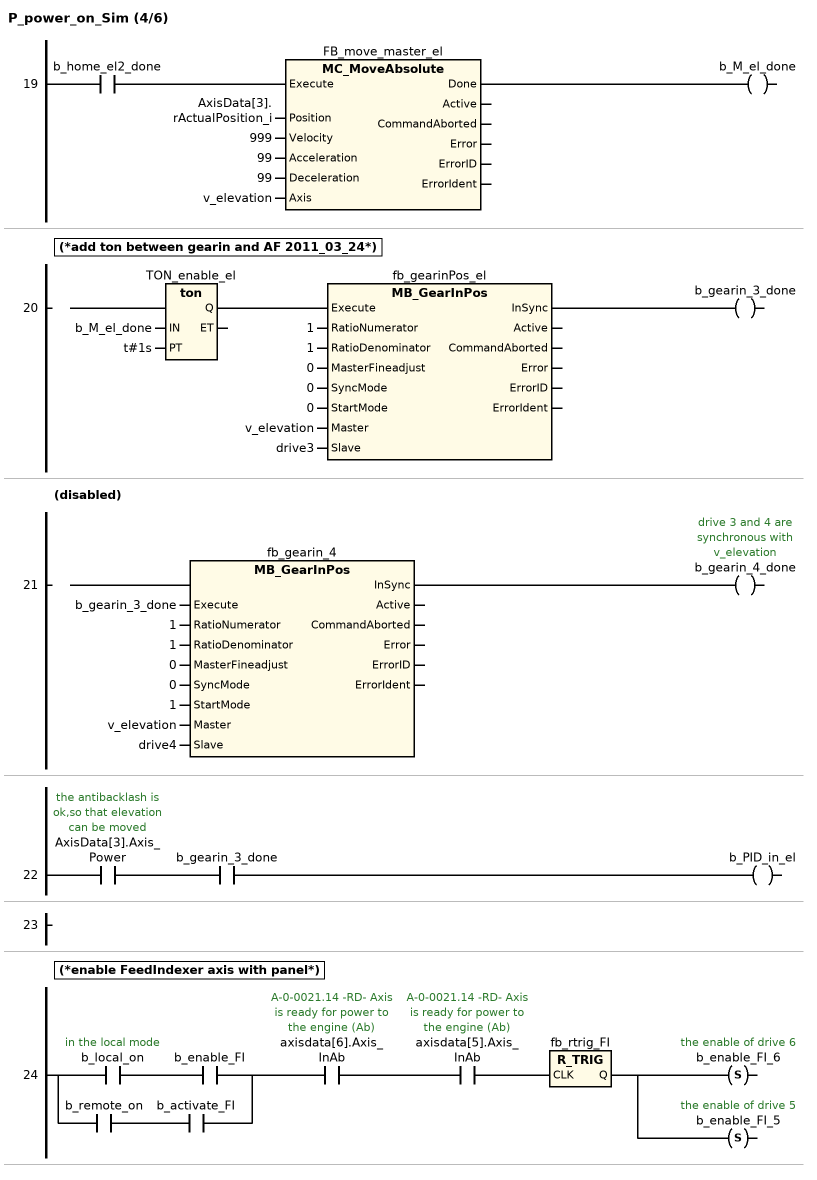
// NETWORK 19
//   AxisData[3].rActualPosition_i: A-0-0100 -RD- Actual position
//   v_elevation: Virtual axis "v_elevation" with axis number 8
FB_move_master_el(
    Execute := b_home_el2_done,
    Position := AxisData[3].rActualPosition_i,
    Velocity := 999,
    Acceleration := 99,
    Deceleration := 99,
    Axis := v_elevation); // MC_MoveAbsolute
b_M_el_done := FB_move_master_el.Done;

// NETWORK 20
//   fb_gearinPos_el: add 2011 06 09 to delete 1sec delay
//   v_elevation: Virtual axis "v_elevation" with axis number 8
//   drive3: Real axis "Drive3" with axis number 3
// label: (*add ton between gearin and AF 2011_03_24*)
TON_enable_el(IN := b_M_el_done, PT := t#1s); // ton
fb_gearinPos_el(
    Execute := TON_enable_el.Q,
    RatioNumerator := 1,
    RatioDenominator := 1,
    MasterFineadjust := 0,
    SyncMode := 0,
    StartMode := 0,
    Master := v_elevation,
    Slave := drive3); // MB_GearInPos
b_gearin_3_done := fb_gearinPos_el.InSync;

// NETWORK 21 (disabled)
//   v_elevation: Virtual axis "v_elevation" with axis number 8
//   drive4: Real axis "Drive4" with axis number 4
//   b_gearin_4_done: drive 3 and 4 are synchronous with v_elevation
// fb_gearin_4(
//     Execute := b_gearin_3_done,
//     RatioNumerator := 1,
//     RatioDenominator := 1,
//     MasterFineadjust := 0,
//     SyncMode := 0,
//     StartMode := 1,
//     Master := v_elevation,
//     Slave := drive4); // MB_GearInPos
// b_gearin_4_done := fb_gearin_4.InSync;

// NETWORK 22
//   AxisData[3].Axis_Power: the antibacklash is ok,so that elevation can be moved
b_PID_in_el := AxisData[3].Axis_Power AND b_gearin_3_done;

// NETWORK 23

// NETWORK 24
//   b_local_on: in the local mode
//   axisdata[6].Axis_InAb: A-0-0021.14 -RD- Axis is ready for power to the engine (Ab)
//   axisdata[5].Axis_InAb: A-0-0021.14 -RD- Axis is ready for power to the engine (Ab)
//   b_enable_FI_6: the enable of drive 6
//   b_enable_FI_5: the enable of drive 5
// label: (*enable FeedIndexer axis with panel*)
fb_rtrig_FI(CLK := (b_local_on AND b_enable_FI OR b_remote_on AND b_activate_FI) AND axisdata[6].Axis_InAb AND axisdata[5].Axis_InAb); // R_TRIG
b_enable_FI_6 S= fb_rtrig_FI.Q;
b_enable_FI_5 S= fb_rtrig_FI.Q;

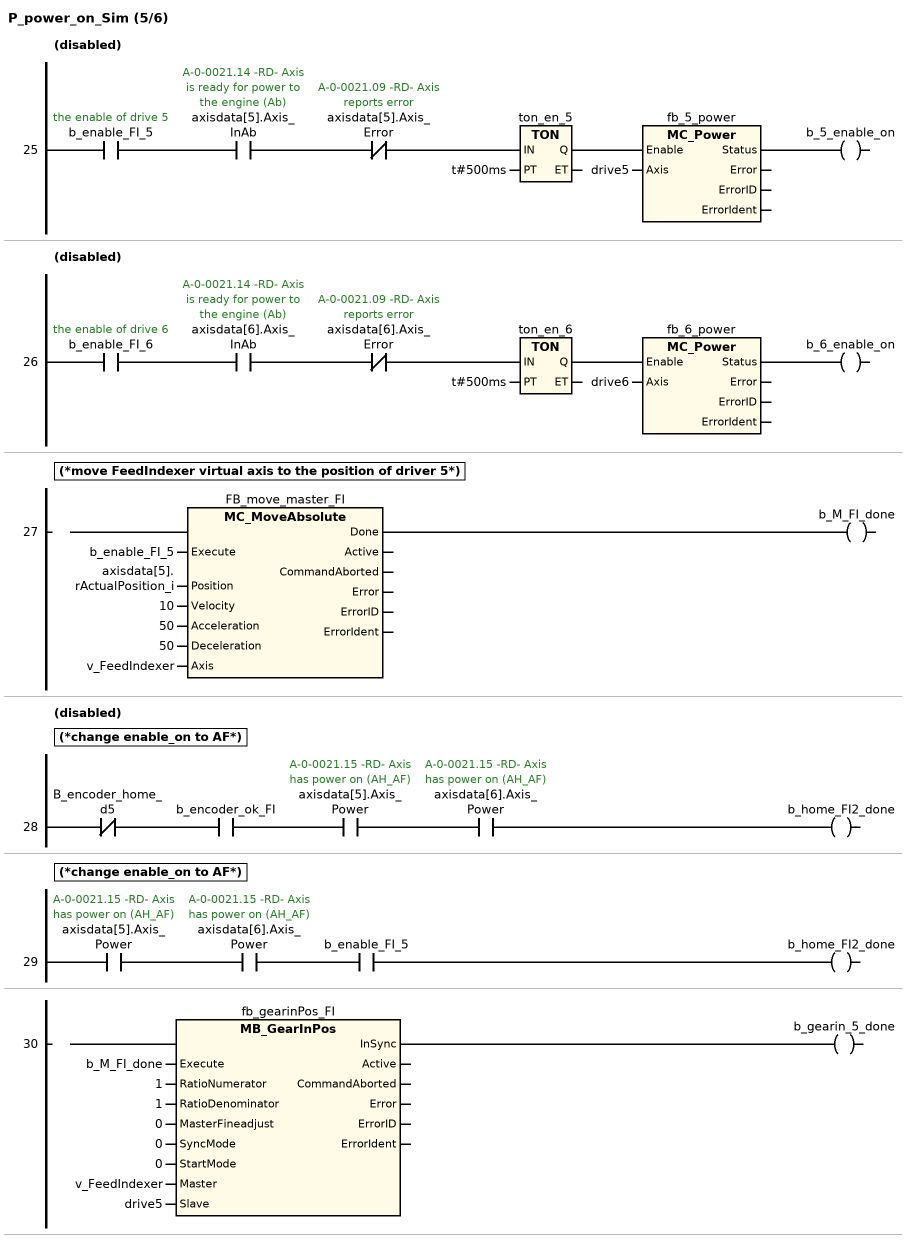
// NETWORK 25 (disabled)
//   b_enable_FI_5: the enable of drive 5
//   axisdata[5].Axis_InAb: A-0-0021.14 -RD- Axis is ready for power to the engine (Ab)
//   axisdata[5].Axis_Error: A-0-0021.09 -RD- Axis reports error
//   drive5: Real axis "Drive5" with axis number 5
// ton_en_5(IN := b_enable_FI_5 AND axisdata[5].Axis_InAb AND NOT axisdata[5].Axis_Error, PT := t#500ms); // TON
// fb_5_power(Enable := ton_en_5.Q, Axis := drive5); // MC_Power
// b_5_enable_on := fb_5_power.Status;

// NETWORK 26 (disabled)
//   b_enable_FI_6: the enable of drive 6
//   axisdata[6].Axis_InAb: A-0-0021.14 -RD- Axis is ready for power to the engine (Ab)
//   axisdata[6].Axis_Error: A-0-0021.09 -RD- Axis reports error
//   drive6: Real axis "Drive6" with axis number 6
// ton_en_6(IN := b_enable_FI_6 AND axisdata[6].Axis_InAb AND NOT axisdata[6].Axis_Error, PT := t#500ms); // TON
// fb_6_power(Enable := ton_en_6.Q, Axis := drive6); // MC_Power
// b_6_enable_on := fb_6_power.Status;

// NETWORK 27
//   axisdata[5].rActualPosition_i: A-0-0100 -RD- Actual position
//   v_FeedIndexer: Virtual axis "v_polarization" with axis number 9
// label: (*move FeedIndexer virtual axis to the position of driver 5*)
FB_move_master_FI(
    Execute := b_enable_FI_5,
    Position := axisdata[5].rActualPosition_i,
    Velocity := 10,
    Acceleration := 50,
    Deceleration := 50,
    Axis := v_FeedIndexer); // MC_MoveAbsolute
b_M_FI_done := FB_move_master_FI.Done;

// NETWORK 28 (disabled)
//   axisdata[5].Axis_Power: A-0-0021.15 -RD- Axis has power on (AH_AF)
//   axisdata[6].Axis_Power: A-0-0021.15 -RD- Axis has power on (AH_AF)
// label: (*change enable_on to AF*)
// b_home_FI2_done := NOT B_encoder_home_d5 AND b_encoder_ok_FI AND axisdata[5].Axis_Power AND axisdata[6].Axis_Power;

// NETWORK 29
//   axisdata[5].Axis_Power: A-0-0021.15 -RD- Axis has power on (AH_AF)
//   axisdata[6].Axis_Power: A-0-0021.15 -RD- Axis has power on (AH_AF)
// label: (*change enable_on to AF*)
b_home_FI2_done := axisdata[5].Axis_Power AND axisdata[6].Axis_Power AND b_enable_FI_5;

// NETWORK 30
//   v_FeedIndexer: Virtual axis "v_polarization" with axis number 9
//   drive5: Real axis "Drive5" with axis number 5
fb_gearinPos_FI(
    Execute := b_M_FI_done,
    RatioNumerator := 1,
    RatioDenominator := 1,
    MasterFineadjust := 0,
    SyncMode := 0,
    StartMode := 0,
    Master := v_FeedIndexer,
    Slave := drive5); // MB_GearInPos
b_gearin_5_done := fb_gearinPos_FI.InSync;

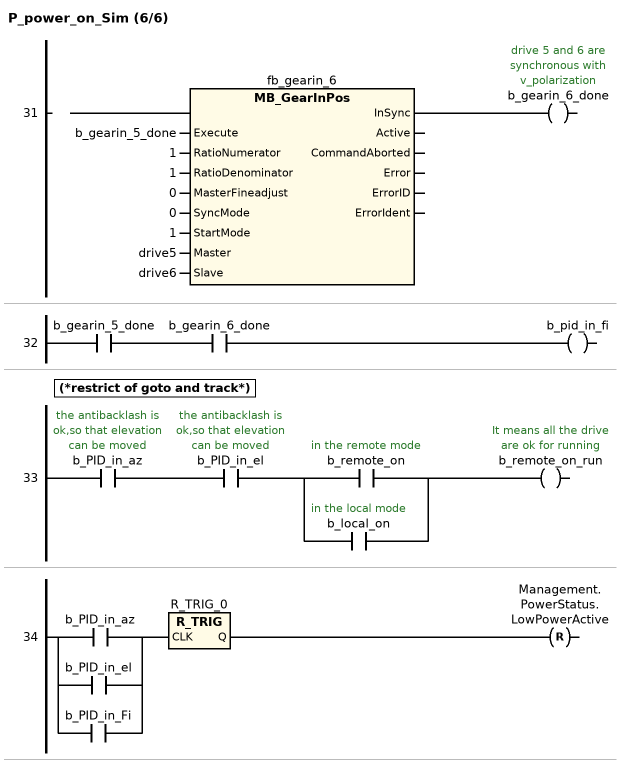
// NETWORK 31
//   drive5: Virtual axis "v_polarization" with axis number 9
//   drive6: Real axis "Drive6" with axis number 6
//   b_gearin_6_done: drive 5 and 6 are synchronous with v_polarization
fb_gearin_6(
    Execute := b_gearin_5_done,
    RatioNumerator := 1,
    RatioDenominator := 1,
    MasterFineadjust := 0,
    SyncMode := 0,
    StartMode := 1,
    Master := drive5,
    Slave := drive6); // MB_GearInPos
b_gearin_6_done := fb_gearin_6.InSync;

// NETWORK 32
b_pid_in_fi := b_gearin_5_done AND b_gearin_6_done;

// NETWORK 33
//   b_PID_in_az: the antibacklash is ok,so that elevation can be moved
//   b_PID_in_el: the antibacklash is ok,so that elevation can be moved
//   b_remote_on: in the remote mode
//   b_local_on: in the local mode
//   b_remote_on_run: It means all the drive are ok for running
// label: (*restrict of goto and track*)
b_remote_on_run := b_PID_in_az AND b_PID_in_el AND (b_remote_on OR b_local_on);

// NETWORK 34
R_TRIG_0(CLK := b_PID_in_az OR b_PID_in_el OR b_PID_in_Fi); // R_TRIG
Management.PowerStatus.LowPowerActive R= R_TRIG_0.Q;

END_PROGRAM

// IndraMotionMlc1/Application/POUs/TCP/P_UDP_with_DAM
(*This program is built for UDP communication, receive the message from CSIRO,deal with the commands,and send the reply to CSIRO*)
PROGRAM P_UDP_with_DAM
VAR
(*<<<<<<<<<<<<<<<<<<<<<<<<<<<<<<<<<<<<<<<<<<<>>>>>>>>>>>>>>>>>>>>>>>>>>>>>>>>>>>>>*)
	b_receiving :BOOL;
	b_receiving_1 :BOOL;
	b_receiving_2 :BOOL;
	b_receiving_3 :BOOL;
	b_commanding: BOOL;
	b_commanding_1: BOOL;
	b_commanding_2: BOOL;
	b_commanding_3: BOOL;
	b_sending: BOOL;
	b_sending_1: BOOL;
	b_sending_2: BOOL;
	b_sending_3: BOOL;
	
(*<<<<<<<<<<<<<<<<<<<<<<<<<<<<<<<<<<<<<<<<<<<CONNECTION>>>>>>>>>>>>>>>>>>>>>>>>>>>>>>>>>>>>>*)
	UDPConnection_1: IL_UDPSocketAsync;
	UDPConnection_2: IL_UDPSocketAsync;
	UDPConnection_3: IL_UDPSocketAsync;
	b_Server_Enable: BOOL:=TRUE;(*the enable of IL_TCPConnectionAsync*)
	b_Server_Enable_1: BOOL:=TRUE;(*the enable of IL_TCPConnectionAsync*)
	b_Server_Enable_2: BOOL:=TRUE;(*the enable of IL_TCPConnectionAsync*)
	b_Server_Enable_3: BOOL:=TRUE;(*the enable of IL_TCPConnectionAsync*)
	di_Socket: DINT;(*the socket number*)
	di_Socket_1: DINT;(*the socket number*)
	di_Socket_2: DINT;(*the socket number*)
	di_Socket_3: DINT;(*the socket number*)
	strIP: STRING;
	b_Connection_done: BOOL;
	b_Connection_done_1: BOOL;
	b_Connection_done_2: BOOL;
	b_Connection_done_3: BOOL;
(*<<<<<<<<<<<<<<<<<<<<<<<<<<<<<<<<<<<<<<<<<<<RECEIVE>>>>>>>>>>>>>>>>>>>>>>>>>>>>>>>>>>>>>*)
	UDPRecv_1: IL_UDPRecvfromAsync;
	UDPRecv_2: IL_UDPRecvfromAsync;
	UDPRecv_3: IL_UDPRecvfromAsync;
	b_Recv_enable: BOOL;
	b_Recv_enable_1: BOOL;
	b_Recv_enable_2: BOOL;
	b_Recv_enable_3: BOOL;
	b_Recv_done: BOOL;
	b_Recv_done_1: BOOL;
	b_Recv_done_2: BOOL;
	b_Recv_done_3: BOOL;
	str_Recv: STRING(255);
	str_Recv_1: ARRAY [1..200] OF BYTE;
	str_Recv_2: ARRAY [1..200] OF BYTE;
	str_Recv_3: ARRAY [1..200] OF BYTE;
	//fb_crc16 : CRC16_MODBUS;
	di_ReceivedBytes: DINT;
	di_ReceivedBytes_1: DINT;
	di_ReceivedBytes_2: DINT;
	di_ReceivedBytes_3: DINT;
(*<<<<<<<<<<<<<<<<<<<<<<<<<<<<<<<<<<<<<<<<<<<<SEND>>>>>>>>>>>>>>>>>>>>>>>>>>>>>>>>>>>>>*)
	UDPSend_1: IL_UDPSendtoAsync;
	UDPSend_2: IL_UDPSendtoAsync;
	UDPSend_3: IL_UDPSendtoAsync;
	b_Send_enable: BOOL;
	b_Send_enable_1: BOOL;
	b_Send_enable_2: BOOL;
	b_Send_enable_3: BOOL;
	b_Send_done: BOOL;
	b_Send_done_1: BOOL;
	b_Send_done_2: BOOL;
	b_Send_done_3: BOOL;
	str_Send: STRING(1000);
	str_Send_1: ARRAY [1..8] OF BYTE;
	str_Send_2: ARRAY [1..8] OF BYTE;
	str_Send_3: ARRAY [1..8] OF BYTE;
	di_SentBytes: DINT;
	di_SentBytes_1: DINT;
	di_SentBytes_2: DINT;
	di_SentBytes_3: DINT;
	
	di_SentBytesLen_1: UINT;
	di_SentBytesLen_2: UINT;
	di_SentBytesLen_3: UINT;

(*add the function of close TCP function*)
	fb_tcp_close: IL_UDPCloseAsync;
	fb_udp_close_1: IL_UDPCloseAsync;
	fb_udp_close_2: IL_UDPCloseAsync;
	fb_udp_close_3: IL_UDPCloseAsync;
	B_TCP_close: BOOL;
	B_TCP_close_1: BOOL;
	B_TCP_close_2: BOOL;
	B_TCP_close_3: BOOL;
	b_TCP_close_done: BOOL;
	b_TCP_close_done_1: BOOL;
	b_TCP_close_done_2: BOOL;
	b_TCP_close_done_3: BOOL;
	b_Recv_active: BOOL;
	b_Recv_active_1: BOOL;
	b_Recv_active_2: BOOL;
	b_Recv_active_3: BOOL;
	i_counter_udp1:INT;
	i_counter_udp2:INT;
	i_counter_udp3:INT;

	str_concat: ARRAY[1..40] OF STRING(1000);(*数组及其类型的定义*)	
	str_concat_1: ARRAY[1..40] OF BYTE;(*数组及其类型的定义*)
	str_concat_2: ARRAY[1..40] OF BYTE;(*数组及其类型的定义*)
	str_concat_3: ARRAY[1..40] OF BYTE;(*数组及其类型的定义*)
	Counter: INT;
	bWaiting4Connection: BOOL;
	bWaiting4Connection_1: BOOL;
	bWaiting4Connection_2: BOOL;
	bWaiting4Connection_3: BOOL;
	bConnError: BOOL;
	bConnError_1: BOOL;
	bConnError_2: BOOL;
	bConnError_3: BOOL;
	diConnError: ERROR_CODE;
	diConnError_1: ERROR_CODE;
	diConnError_2: ERROR_CODE;
	diConnError_3: ERROR_CODE;
	ConnectError: ERROR_STRUCT;
	ConnectError_1: ERROR_STRUCT;
	ConnectError_2: ERROR_STRUCT;
	ConnectError_3: ERROR_STRUCT;
	i_counter_1s: INT:=0;	
	i_count:INT;
	
	reply_count: DINT;
	index: BYTE;
	
	dam1_data1 : LREAL;
	dam1_data2 : LREAL;
	dam1_data3 : LREAL;
	dam1_data4 : LREAL;
	dam1_data5 : LREAL;
	dam1_data6 : LREAL;
	dam1_data7 : LREAL;
	dam1_data8 : LREAL;
	dam1_data9 : LREAL;
	dam1_data10 : LREAL;
	dam1_data11 : LREAL;
	dam1_data12 : LREAL;
	

	
	dam3_data1 : REAL;
	dam3_data2 : REAL;
	dam3_data3 : REAL;
	dam3_data4 : REAL;
	dam3_data5 : REAL;
	dam3_data6 : REAL;
	dam3_data7 : REAL;
	dam3_data8 : REAL;
	dam3_data9 : REAL;
	dam3_data10 : REAL;
	dam3_data11 : REAL;
	dam3_data12 : REAL;
	dam3_data13 : REAL;
	dam3_data14 : REAL;
	dam3_data15 : REAL;
	dam3_data16 : REAL;
	dam3_data17 : REAL;
	dam3_data18 : REAL;
	dam3_data19 : REAL;
	dam3_data20 : REAL;
	dam3_data21 : REAL;
	dam3_data22 : REAL;
	dam3_data23 : REAL;
	dam3_data24 : REAL;
	dam3_data25 : REAL;
	dam3_data26 : REAL;
	dam3_data27 : REAL;
	dam3_data28 : REAL;
	fb_crc16_modbus: CRC16_MODBUS;
	
	a_phase_current : REAL;
	b_phase_current : REAL;
	c_phase_current : REAL;
	a_phase_voltage : REAL;
	b_phase_voltage : REAL;
	c_phase_voltage : REAL;
	ab_line_voltage : REAL;
	bc_line_voltage : REAL;
	ca_line_voltage : REAL;
	a_phase_activepower : REAL;
	b_phase_activepower : REAL;
	c_phase_activepower : REAL;
	a_phase_reactivepower : REAL;
	b_phase_reactivepower : REAL;
	c_phase_reactivepower : REAL;
	a_phase_apparentpower : REAL;
	b_phase_apparentpower : REAL;
	c_phase_apparentpower : REAL;
	a_phase_powerfactor : REAL;
	b_phase_powerfactor : REAL;
	c_phase_powerfactor : REAL;
	a_phase_frequency : REAL;
	b_phase_frequency : REAL;
	c_phase_frequency : REAL;
	total_activepower : REAL;
	total_reactivepower : REAL;
	total_apparentpower : REAL;
	total_powerfactor : REAL;
	
	
	X_Axis_Tile_Monitor : LREAL;
	Y_Axis_Tile_Monitor : LREAL;
	Temp_Tile_Monitor : LREAL;
	
	HumidEMISC_Outlet: LREAL;
END_VAR


reply_count:=reply_count+1;

IF reply_count < 0 OR reply_count >= 40 THEN	
	reply_count:=0;
END_IF

IF reply_count >= 0 AND reply_count < 10 THEN 
(*<<<<<<<<<<<<<<<<<<<<<<<<<<<<<concatenate STR_DAM1>>>>>>>>>>>>>>>>>>>>>>>>>>>>>>>>>>>>>>>>>>>>>>>>>>>>>>>*)
	str_concat_1[1] := 16#01;	//设备地址1
	str_concat_1[2] := 16#04;	//功能码
	str_concat_1[3] := 16#00;	//寄存器地址1
	str_concat_1[4] := 16#00;	//寄存器地址2
	str_concat_1[5] := 16#00;	//寄存器数量1
	str_concat_1[6] := 16#10;	//寄存器地址2
	fb_crc16_modbus(str_Message:= str_concat_1, str_Len:= 6, crc16=> );		//计算CRC校验
	str_concat_1[7] := WORD_TO_BYTE(fb_crc16_modbus.crc16 AND 16#00FF);
	str_concat_1[8] := WORD_TO_BYTE(SHR(fb_crc16_modbus.crc16,8) AND 16#00FF);
	FOR index:=1 TO 8 BY 1 DO
		str_send_1[index] := 16#00;
	END_FOR
	FOR index:=1 TO 8 BY 1 DO
		str_send_1[index] := str_concat_1[index];
	END_FOR
	di_SentBytesLen_1 := 8;
ELSIF reply_count >= 10 AND reply_count < 20 THEN
(*<<<<<<<<<<<<<<<<<<<<<<<<<<<<<concatenate STR_DAM2>>>>>>>>>>>>>>>>>>>>>>>>>>>>>>>>>>>>>>>>>>>>>>>>>>>>>>>*)
	str_concat_1[1] := 16#02;	//设备地址1
	str_concat_1[2] := 16#04;	//功能码
	str_concat_1[3] := 16#00;	//寄存器地址1
	str_concat_1[4] := 16#00;	//寄存器地址2
	str_concat_1[5] := 16#00;	//寄存器数量1
	str_concat_1[6] := 16#03;	//寄存器地址2
	fb_crc16_modbus(str_Message:= str_concat_1, str_Len:= 6, crc16=> );		//计算CRC校验
	str_concat_1[7] := WORD_TO_BYTE(fb_crc16_modbus.crc16 AND 16#00FF);
	str_concat_1[8] := WORD_TO_BYTE(SHR(fb_crc16_modbus.crc16,8) AND 16#00FF);
	FOR index:=1 TO 8 BY 1 DO
		str_send_1[index] := 16#00;
	END_FOR
	FOR index:=1 TO 8 BY 1 DO
		str_send_1[index] := str_concat_1[index];
	END_FOR
	di_SentBytesLen_1 := 8;
ELSIF reply_count >= 20 AND reply_count < 30 THEN
(*<<<<<<<<<<<<<<<<<<<<<<<<<<<<<concatenate STR_DAM2>>>>>>>>>>>>>>>>>>>>>>>>>>>>>>>>>>>>>>>>>>>>>>>>>>>>>>>*)
	str_concat_1[1] := 16#03;	//设备地址1
	str_concat_1[2] := 16#04;	//功能码
	str_concat_1[3] := 16#00;	//寄存器地址1
	str_concat_1[4] := 16#00;	//寄存器地址2
	str_concat_1[5] := 16#00;	//寄存器数量1
	str_concat_1[6] := 16#06;	//寄存器地址2
	fb_crc16_modbus(str_Message:= str_concat_1, str_Len:= 6, crc16=> );		//计算CRC校验
	str_concat_1[7] := WORD_TO_BYTE(fb_crc16_modbus.crc16 AND 16#00FF);
	str_concat_1[8] := WORD_TO_BYTE(SHR(fb_crc16_modbus.crc16,8) AND 16#00FF);
	FOR index:=1 TO 8 BY 1 DO
		str_send_1[index] := 16#00;
	END_FOR
	FOR index:=1 TO 8 BY 1 DO
		str_send_1[index] := str_concat_1[index];
	END_FOR
	di_SentBytesLen_1 := 8;
ELSE
(*<<<<<<<<<<<<<<<<<<<<<<<<<<<<<concatenate STR_DAM3>>>>>>>>>>>>>>>>>>>>>>>>>>>>>>>>>>>>>>>>>>>>>>>>>>>>>>>*)
	str_concat_1[1] := 16#03;	//设备地址1
	str_concat_1[2] := 16#04;	//功能码
	str_concat_1[3] := 16#00;	//寄存器地址1
	str_concat_1[4] := 16#27;	//寄存器地址2
	str_concat_1[5] := 16#00;	//寄存器数量1
	str_concat_1[6] := 16#0D;	//寄存器地址2
	fb_crc16_modbus(str_Message:= str_concat_1, str_Len:= 6, crc16=> );		//计算CRC校验
	str_concat_1[7] := WORD_TO_BYTE(fb_crc16_modbus.crc16 AND 16#00FF);
	str_concat_1[8] := WORD_TO_BYTE(SHR(fb_crc16_modbus.crc16,8) AND 16#00FF);
	FOR index:=1 TO 8 BY 1 DO
		str_send_1[index] := 16#00;
	END_FOR
	FOR index:=1 TO 8 BY 1 DO
		str_send_1[index] := str_concat_1[index];
	END_FOR	
	di_SentBytesLen_1 := 8;
END_IF
				
(*<<<<<<<<<<<<<<<<<<<<<<<<<<<if TCP is wrong,reset the TCP serve>>>>>>>>>>>>>>>>>>>>>>>>>>>>*)
IF UDPConnection_1.Error=TRUE OR UDPRecv_1.Error=TRUE OR UDPSend_1.Error=TRUE THEN
	b_Server_Enable_1:=FALSE;
	b_Recv_enable_1:=FALSE;
	b_Send_enable_1:=FALSE;
ELSE
	b_Server_Enable_1:=TRUE;
END_IF

IF UDPConnection_2.Error=TRUE OR UDPRecv_2.Error=TRUE OR UDPSend_2.Error=TRUE THEN
	b_Server_Enable_2:=FALSE;
	b_Recv_enable_2:=FALSE;
	b_Send_enable_2:=FALSE;
ELSE
	b_Server_Enable_2:=TRUE;
END_IF

P_UDP_with_DAM.Async_TCP();
P_UDP_with_DAM.A_RECV();
P_UDP_with_DAM.A_SEND();
(*<<<<<<<<<<<<<<<<<<<<<<<<<<<if TCP server is connected,a cycle is executed>>>>>>>>>>>>>>>>>>>>>>>>>>>>>>>>>>>>>>>>>>>>>*)
IF b_Connection_done_1=TRUE THEN
	IF  b_receiving_1=FALSE AND b_sending_1=FALSE AND b_Send_enable_1=FALSE THEN
		b_Send_enable_1:=TRUE;(*open send fuction*)
		P_UDP_with_DAM.A_SEND();
		b_sending_1:=TRUE;
	END_IF;
	
(*<<<<<<<<<<<<<<<<<<<<<<<<<<<send message>>>>>>>>>>>>>>>>>>>>>>>>>>>>>>>>>>>>>>>>>>>>>>>>>*)
	IF b_Send_done_1=TRUE AND b_sending_1=TRUE AND b_receiving_1=FALSE THEN
		b_Send_enable_1:=FALSE;
		P_UDP_with_DAM.A_SEND();
		b_sending_1:=FALSE;
		b_receiving_1:=TRUE;
		i_counter_udp1 := 0;
	END_IF;
	
(*<<<<<<<<<<<<<<<<<<<<<<<<<<<<<<<<<<<<<<<<<<<<<<<<<receive message>>>>>>>>>>>>>>>>>>>>>>>>>>>>>>>>>>>>>>>>>>>>>>>>>>>>>>>*)
	IF b_sending_1=FALSE AND b_receiving_1=TRUE THEN
		b_Recv_enable_1:=TRUE;
		P_UDP_with_DAM.A_RECV();
		i_counter_udp1 := i_counter_udp1 + 1;
	END_IF;
	
(*<<<<<<<<<<<<<<<<<<<<<<<<<<<<<<<<<<<<<<<<<<<<<<<<<not receive message>>>>>>>>>>>>>>>>>>>>>>>>>>>>>>>>>>>>>>>>>>>>>>>>>>>>>>>*)	
	IF b_sending_1=FALSE AND b_receiving_1=TRUE AND i_counter_udp1>10 THEN
		b_Recv_enable_1:=FALSE;
		b_receiving_1:=FALSE;
		i_counter_udp1 := 0;
	END_IF;
	
(*<<<<<<<<<<<<<<<<<<<<<<<<<<<recieveing message>>>>>>>>>>>>>>>>>>>>>>>>>>>>>>>>>>>>>>>>>>>>>>>>>*)
	IF b_Recv_done_1=TRUE AND b_receiving_1=TRUE THEN
		
		IF str_Recv_1[1] = 16#01 AND str_Recv_1[3] = 16#20 THEN
			
			TempEMISC_Outlet := WORD_TO_LREAL(BYTE_TO_WORD(str_Recv_1[16]) * 256 + BYTE_TO_WORD(str_Recv_1[17])) / 65535 * 165 - 40;
			HumidEMISC_Outlet := WORD_TO_LREAL(BYTE_TO_WORD(str_Recv_1[18]) * 256 + BYTE_TO_WORD(str_Recv_1[19])) / 65535 * 100;
			TempPSC_Inlet := WORD_TO_LREAL(BYTE_TO_WORD(str_Recv_1[20]) * 256 + BYTE_TO_WORD(str_Recv_1[21])) / 65535 * 165 - 40;
			HumidPSC_Inlet := WORD_TO_LREAL(BYTE_TO_WORD(str_Recv_1[22]) * 256 + BYTE_TO_WORD(str_Recv_1[23])) / 65535 * 100;
			TempPSC_Outlet := WORD_TO_LREAL(BYTE_TO_WORD(str_Recv_1[24]) * 256 + BYTE_TO_WORD(str_Recv_1[25])) / 65535 * 165 - 40;
			HumidPSC_Outlet := WORD_TO_LREAL(BYTE_TO_WORD(str_Recv_1[26]) * 256 + BYTE_TO_WORD(str_Recv_1[27])) / 65535 * 100;
			TempDriveCab := WORD_TO_LREAL(BYTE_TO_WORD(str_Recv_1[28]) * 256 + BYTE_TO_WORD(str_Recv_1[29])) / 65535 * 100 - 20;
			HumidDriveCab := WORD_TO_LREAL(BYTE_TO_WORD(str_Recv_1[30]) * 256 + BYTE_TO_WORD(str_Recv_1[31])) / 65535 * 100;
			TempDriveCab_Up := WORD_TO_LREAL(BYTE_TO_WORD(str_Recv_1[32]) * 256 + BYTE_TO_WORD(str_Recv_1[33])) / 65535 * 100 - 20;
			HumidDriveCab_Up := WORD_TO_LREAL(BYTE_TO_WORD(str_Recv_1[34]) * 256 + BYTE_TO_WORD(str_Recv_1[35])) / 65535 * 100;			 

			
		ELSIF str_Recv_1[1] = 16#02 AND str_Recv_1[3] = 16#06 THEN
			
			Pedestal_temp_1 := WORD_TO_REAL(BYTE_TO_WORD(str_Recv_1[4]) * 256 + BYTE_TO_WORD(str_Recv_1[5])) / 65535 * 200 - 50;
			Pedestal_temp_2 := WORD_TO_REAL(BYTE_TO_WORD(str_Recv_1[6]) * 256 + BYTE_TO_WORD(str_Recv_1[7])) / 65535 * 200 - 50;
			Pedestal_temp_3 := WORD_TO_REAL(BYTE_TO_WORD(str_Recv_1[8]) * 256 + BYTE_TO_WORD(str_Recv_1[9])) / 65535 * 200 - 50;
			
		ELSIF str_Recv_1[1] = 16#03 AND str_Recv_1[3] =16#0C THEN
			
			CurrentPh1 := WORD_TO_LREAL(BYTE_TO_WORD(str_Recv_1[4]) * 256 + BYTE_TO_WORD(str_Recv_1[5])) / 65535 * 100;
			CurrentPh2 := WORD_TO_LREAL(BYTE_TO_WORD(str_Recv_1[6]) * 256 + BYTE_TO_WORD(str_Recv_1[7])) / 65535 * 100;
			CurrentPh3 := WORD_TO_LREAL(BYTE_TO_WORD(str_Recv_1[8]) * 256 + BYTE_TO_WORD(str_Recv_1[9])) / 65535 * 100;
			VoltagePh1 := WORD_TO_LREAL(BYTE_TO_WORD(str_Recv_1[10]) * 256 + BYTE_TO_WORD(str_Recv_1[11])) / 65535 * 1000;
			VoltagePh2 := WORD_TO_LREAL(BYTE_TO_WORD(str_Recv_1[12]) * 256 + BYTE_TO_WORD(str_Recv_1[13])) / 65535 * 1000;
			VoltagePh3 := WORD_TO_LREAL(BYTE_TO_WORD(str_Recv_1[14]) * 256 + BYTE_TO_WORD(str_Recv_1[15])) / 65535 * 1000;
		
		ELSIF str_Recv_1[1] = 16#03 AND str_Recv_1[3] =16#1A THEN
		
			FrequencyPh1 := WORD_TO_LREAL(BYTE_TO_WORD(str_Recv_1[4]) * 256 + BYTE_TO_WORD(str_Recv_1[5])) / 65535 * 65;
			FrequencyPh2 := WORD_TO_LREAL(BYTE_TO_WORD(str_Recv_1[6]) * 256 + BYTE_TO_WORD(str_Recv_1[7])) / 65535 * 65;
			FrequencyPh3 := WORD_TO_LREAL(BYTE_TO_WORD(str_Recv_1[8]) * 256 + BYTE_TO_WORD(str_Recv_1[9])) / 65535 * 65;
			
			ActivePowerConsumption := WORD_TO_LREAL(BYTE_TO_WORD(str_Recv_1[10]) * 256 + BYTE_TO_WORD(str_Recv_1[11])) / 65535 * 600000 - 300000;
			ReactivePowerConsumption := WORD_TO_LREAL(BYTE_TO_WORD(str_Recv_1[12]) * 256 + BYTE_TO_WORD(str_Recv_1[13])) / 65535 * 600000 - 300000;
			ApparentPowerConsumption := WORD_TO_LREAL(BYTE_TO_WORD(str_Recv_1[14]) * 256 + BYTE_TO_WORD(str_Recv_1[15])) / 65535 * 600000 - 300000;

		
			PowerFactor := WORD_TO_LREAL(BYTE_TO_WORD(str_Recv_1[28]) * 256 + BYTE_TO_WORD(str_Recv_1[29])) / 65535 * 2 - 1;
	
		END_IF;

		b_Recv_enable_1:=FALSE;
		P_UDP_with_DAM.A_RECV();
		b_receiving_1:=FALSE;
		i_counter_udp1 := 0;
	END_IF;
	
	IF b_Recv_done_1=TRUE  THEN
		b_Recv_enable_1:=FALSE;
		P_UDP_with_DAM.A_RECV();
	END_IF;
(*<<<<<<<<<<<<<<<<<<<<<<<<<<<<<<<<<<<<<<<<<<<<<If not conected,then reset receive and send function>>>>>>>>>>>>>>>>>>>>>>>>>>>>>>>>>>>>>>>>>>>>>>>>>>>>>>>*)
ELSE
	b_receiving_1:=FALSE;
	b_sending_1:=FALSE;
	b_Recv_enable_1:=FALSE;
	b_send_enable_1:=FALSE;
END_IF;

(*Tilt Sensor Receiving Data*)
IF b_Connection_done_2=TRUE THEN
	IF  b_receiving_2=FALSE AND b_sending_2=FALSE AND b_Recv_enable_2=FALSE THEN
		b_Recv_enable_2:=TRUE;(*open receive fuction*)
		P_UDP_with_DAM.A_RECV();
		b_receiving_2:=TRUE;
	END_IF;
	
	IF b_Recv_done_2=TRUE AND b_receiving_2=TRUE THEN
		Pointing.Status.TiltXRaw_mV_One:= WORD_TO_LREAL(BYTE_TO_WORD(str_Recv_2[22]) * 256 + BYTE_TO_WORD(str_Recv_2[23]));
		Pointing.Status.TiltYRaw_mV_One := WORD_TO_LREAL(BYTE_TO_WORD(str_Recv_2[24]) * 256 + BYTE_TO_WORD(str_Recv_2[25]));
		Pointing.Status.TiltTemp_One := WORD_TO_LREAL(BYTE_TO_WORD(str_Recv_2[26]) * 256 + BYTE_TO_WORD(str_Recv_2[27]));
		X_Axis_Tile_Monitor := WORD_TO_LREAL(BYTE_TO_WORD(str_Recv_2[30]) * 256 + BYTE_TO_WORD(str_Recv_2[31]));
		Y_Axis_Tile_Monitor := WORD_TO_LREAL(BYTE_TO_WORD(str_Recv_2[32]) * 256 + BYTE_TO_WORD(str_Recv_2[33]));
		Temp_Tile_Monitor := WORD_TO_LREAL(BYTE_TO_WORD(str_Recv_2[34]) * 256 + BYTE_TO_WORD(str_Recv_2[35]));
	
		b_Recv_enable_2:=FALSE;
		P_UDP_with_DAM.A_RECV();
		b_receiving_2:=FALSE;
	END_IF;
ELSE
	b_receiving_2:=FALSE;
	b_sending_2:=FALSE;
	b_Recv_enable_2:=FALSE;
	b_send_enable_2:=FALSE;
END_IF;

ACTION Async_TCP:
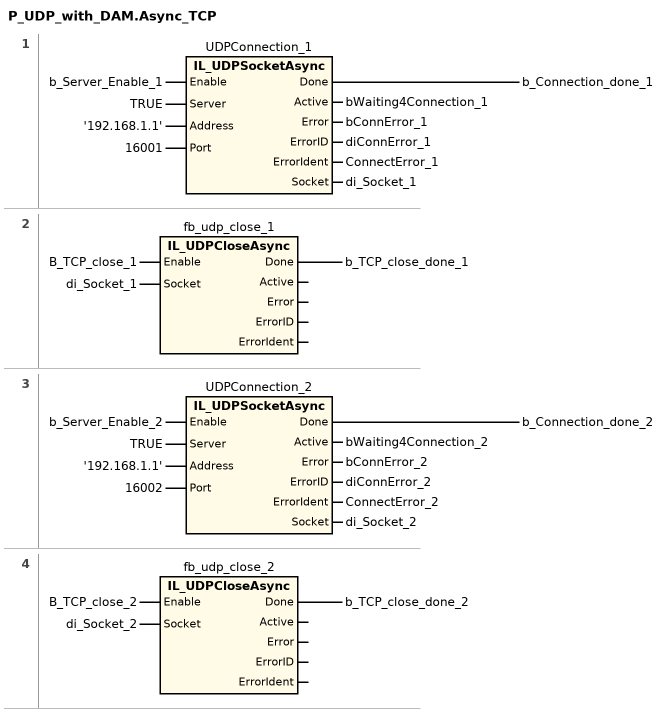
// NETWORK 1
UDPConnection_1(
    Enable := b_Server_Enable_1,
    Server := TRUE,
    Address := '192.168.1.1',
    Port := 16001,
    Active => bWaiting4Connection_1,
    Error => bConnError_1,
    ErrorID => diConnError_1,
    ErrorIdent => ConnectError_1,
    Socket => di_Socket_1); // IL_UDPSocketAsync
b_Connection_done_1 := UDPConnection_1.Done;

// NETWORK 2
fb_udp_close_1(Enable := B_TCP_close_1, Socket := di_Socket_1); // IL_UDPCloseAsync
b_TCP_close_done_1 := fb_udp_close_1.Done;

// NETWORK 3
UDPConnection_2(
    Enable := b_Server_Enable_2,
    Server := TRUE,
    Address := '192.168.1.1',
    Port := 16002,
    Active => bWaiting4Connection_2,
    Error => bConnError_2,
    ErrorID => diConnError_2,
    ErrorIdent => ConnectError_2,
    Socket => di_Socket_2); // IL_UDPSocketAsync
b_Connection_done_2 := UDPConnection_2.Done;

// NETWORK 4
fb_udp_close_2(Enable := B_TCP_close_2, Socket := di_Socket_2); // IL_UDPCloseAsync
b_TCP_close_done_2 := fb_udp_close_2.Done;
END_ACTION

ACTION A_RECV:
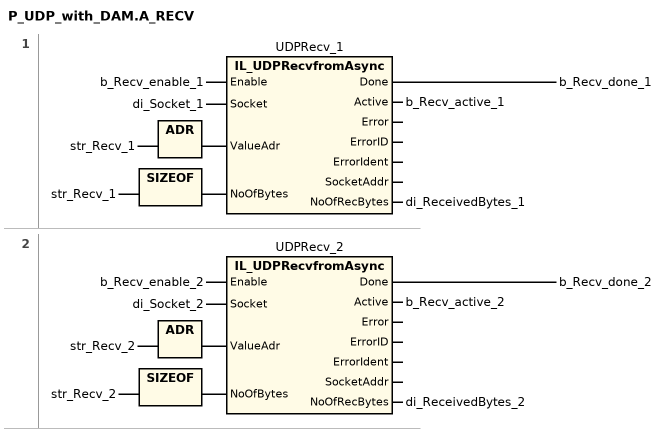
// NETWORK 1
UDPRecv_1(
    Enable := b_Recv_enable_1,
    Socket := di_Socket_1,
    ValueAdr := ADR(str_Recv_1),
    NoOfBytes := SIZEOF(str_Recv_1),
    Active => b_Recv_active_1,
    NoOfRecBytes => di_ReceivedBytes_1); // IL_UDPRecvfromAsync
b_Recv_done_1 := UDPRecv_1.Done;

// NETWORK 2
UDPRecv_2(
    Enable := b_Recv_enable_2,
    Socket := di_Socket_2,
    ValueAdr := ADR(str_Recv_2),
    NoOfBytes := SIZEOF(str_Recv_2),
    Active => b_Recv_active_2,
    NoOfRecBytes => di_ReceivedBytes_2); // IL_UDPRecvfromAsync
b_Recv_done_2 := UDPRecv_2.Done;
END_ACTION

ACTION A_SEND:
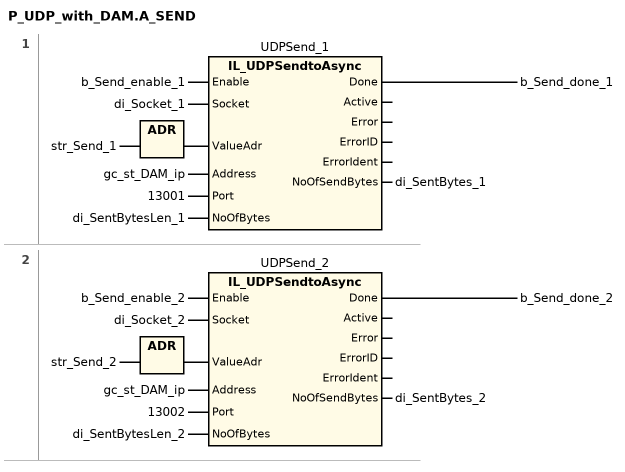
// NETWORK 1
UDPSend_1(
    Enable := b_Send_enable_1,
    Socket := di_Socket_1,
    ValueAdr := ADR(str_Send_1),
    Address := gc_st_DAM_ip,
    Port := 13001,
    NoOfBytes := di_SentBytesLen_1,
    NoOfSendBytes => di_SentBytes_1); // IL_UDPSendtoAsync
b_Send_done_1 := UDPSend_1.Done;

// NETWORK 2
UDPSend_2(
    Enable := b_Send_enable_2,
    Socket := di_Socket_2,
    ValueAdr := ADR(str_Send_2),
    Address := gc_st_DAM_ip,
    Port := 13002,
    NoOfBytes := di_SentBytesLen_2,
    NoOfSendBytes => di_SentBytes_2); // IL_UDPSendtoAsync
b_Send_done_2 := UDPSend_2.Done;
END_ACTION

END_PROGRAM

// IndraMotionMlc1/Application/POUs/TCP/Message/CRC16_MODBUS
FUNCTION_BLOCK CRC16_MODBUS
VAR_INPUT
	str_Message: ARRAY[1..40] OF BYTE;
	str_Len: BYTE;
END_VAR
VAR_OUTPUT
	crc16 : WORD;
END_VAR
VAR
	i : BYTE;
	j : BYTE;
	polynomial : WORD;
	curval : WORD;
	temp : WORD;
END_VAR


temp := 16#FFFF;
polynomial := 16#A001;
FOR i:=1 TO str_Len BY 1 DO
	curval := BYTE_TO_WORD(str_Message[i]);
	FOR j:=1 TO 8 BY 1 DO
		IF ((WORD_TO_BYTE(temp XOR curval) AND 16#01) = 16#01) THEN
			temp := (SHR(temp,1) XOR polynomial);
		ELSE
			temp := SHR(temp,1);			
		END_IF;
		curval := SHR(curval,1);
	END_FOR;
END_FOR;

crc16 := temp;

END_FUNCTION_BLOCK

// IndraMotionMlc1/Application/POUs/TCP/P_GSTAT_K2STAT
(*the program is built for GSTAT and KSTAT,according to ICD*)
PROGRAM P_GSTAT_K2STAT
VAR
(*the transitional variables for GSTAT and KSTAT*)
    STR_GSTAT: STRING(1500);
	STR_K2STAT: STRING(255);
	STR_K4STAT: STRING(255);

(*The function block BLINK generates a pulsating signal.The input consists of ENABLE of the type BOOL, as well as TIMELOW and TIMEHIGH of the type TIME.*)
	fb_blink_diagnos_1: BLINK;
	fb_blink_diagnos_2: BLINK;
	fb_blink_diagnos_3: BLINK;
	fb_blink_diagnos_4: BLINK;
	fb_blink_diagnos_5: BLINK;
	fb_blink_diagnos_6: BLINK;
	fb_blink_diagnos_MLC: BLINK;
(*With the function block "MB_ReadParameter" it is possible to read the current value of a parameter. The return value is DINT*)
	fb_read_brake_1: MB_ReadParameter;
	fb_read_brake_2: MB_ReadParameter;
	fb_read_brake_3: MB_ReadParameter;
	fb_read_brake_4: MB_ReadParameter;
	fb_read_brake_5: MB_ReadParameter;
	fb_read_brake_6: MB_ReadParameter;
(*With the function block "MB_ReadStringParameter" it is possible to read a parameter the operating data of which has the ASCII format (string).*)
	fb_diagnose_1: MB_ReadStringParameter;
	fb_diagnose_2: MB_ReadStringParameter;
	fb_diagnose_3: MB_ReadStringParameter;
	fb_diagnose_4: MB_ReadStringParameter;
	fb_diagnose_5: MB_ReadStringParameter;
	fb_diagnose_6: MB_ReadStringParameter;
	fb_diagnose_MLC: MB_ReadStringParameter;
(*With the function block "MB_ReadRealParameter" it is possible to read the current value of a parameter. The return value is REAL. *)
	FB_readcur1: MB_ReadRealParameter;
	FB_readcur2: MB_ReadRealParameter;
	FB_readcur3: MB_ReadRealParameter;
	FB_readcur4: MB_ReadRealParameter;
	FB_readcur5: MB_ReadRealParameter;
	FB_readcur6: MB_ReadRealParameter;
	fb_temp_1: MB_ReadRealParameter;
	fb_temp_2: MB_ReadRealParameter;
	fb_temp_3: MB_ReadRealParameter;
	fb_temp_4: MB_ReadRealParameter;
	fb_temp_5: MB_ReadRealParameter;
	fb_temp_6: MB_ReadRealParameter;
	fb_read_s189_1: MB_ReadRealParameter;
	fb_read_s189_3: MB_ReadRealParameter;
	fb_read_s189_5: MB_ReadRealParameter;
	FB_readtor1: MB_ReadRealParameter;
	FB_readtor2: MB_ReadRealParameter;
	FB_readtor3: MB_ReadRealParameter;
	FB_readtor4: MB_ReadRealParameter;
	FB_readtor5: MB_ReadRealParameter;
	FB_readtor6: MB_ReadRealParameter;
	FB_temp_1_a: MB_ReadRealParameter;
	FB_temp_2_a: MB_ReadRealParameter;
	FB_temp_3_a: MB_ReadRealParameter;
	FB_temp_4_a: MB_ReadRealParameter;
	FB_temp_5_a: MB_ReadRealParameter;
	FB_temp_6_a: MB_ReadRealParameter;
(*FP_P_0_0539,Holding brake status word *)
	dw_brake_1: DWORD;
	dw_brake_2: DWORD;
	dw_brake_3: DWORD;
	dw_brake_4: DWORD;
	dw_brake_5: DWORD;
	dw_brake_6: DWORD;
(*FP_P_0_0007,Display text of diagnostic message*)
	str_diagnose_MLC: STRING;
	str_diagnose_1: STRING;
	str_diagnose_2: STRING;
	str_diagnose_3: STRING;
	str_diagnose_4: STRING;
	str_diagnose_5: STRING;
	str_diagnose_6: STRING;

(*FP_S_0_0384,Amplifier temperature*)
	r_temp_amp1: REAL;
	r_temp_amp2: REAL;
	r_temp_amp3: REAL;
	r_temp_amp4: REAL;
	r_temp_amp5: REAL;
	r_temp_amp6: REAL;


(*<<<<<<<<<<<<<<<<<<<<<<<<<<<<<<<<<<<<<<<add MLC temperature and operation hour(20100708)>>>>>>>>>>>>>>>>>>>>>>>>>>>>>>>>>>>>>*)
	fb_temp_MLC: MB_ReadRealParameter;
	r_temp_MLC: REAL;(*FP_c_0_0070,Control unit temperature*)
	fb_read_system_status: MB_ReadParameter;
	dw_system_status: DWORD;(*FP_C_0_0023,MC system status,used for temperature warning*)
	fb_read_operation_hour: MB_ReadParameter;

(*the limit for judging whether azimuth following error is too big*)
	r_limit_track_az: REAL;
(*test for limit check*)
	fb_software_limit_1: MB_ReadParameter;
	fb_software_limit_5: MB_ReadParameter;
	fb_software_limit_3: MB_ReadParameter;
	fb_hardware_limit_1: MB_ReadParameter;
	fb_hardware_limit_3: MB_ReadParameter;
	fb_hardware_limit_5: MB_ReadParameter;
	fb_ESTOP_1: MB_ReadParameter;
	fb_ESTOP_3: MB_ReadParameter;
	fb_ESTOP_5: MB_ReadParameter;
	i_software_limit_1: DINT;
	i_software_limit_3: DINT;
	i_software_limit_5: DINT;
	i_hardware_limit_1: DINT;
	i_hardware_limit_3: DINT;
	i_hardware_limit_5: DINT;
	i_ESTOP_1: DINT;
	i_ESTOP_3: DINT;
	i_ESTOP_5: DINT;


	b_azimuth_limit: BOOL;
	b_elevation_limit: BOOL;
	b_FeedIndexer_limit: BOOL;
	fb_readpar_speed_1: MB_ReadRealParameter;
	fb_readpar_speed_3: MB_ReadRealParameter;
	fb_readpar_speed_5: MB_ReadRealParameter;
	
	str_concat: ARRAY[1..40] OF STRING(1500);(*数组及其类型的定义*)	
	Counter: INT;
	FB_readmotorencoder1: MB_ReadRealParameter;
	FB_readmotorencoder2: MB_ReadRealParameter;
	FB_readmotorencoder3: MB_ReadRealParameter;
	FB_readmotorencoder4: MB_ReadRealParameter;
	FB_readmotorencoder5: MB_ReadRealParameter;
	FB_readmotorencoder6: MB_ReadRealParameter;
	r_motorencoder_6: REAL;
	r_motorencoder_5: REAL;
	r_motorencoder_4: REAL;
	r_motorencoder_3: REAL;
	r_motorencoder_2: REAL;
	r_motorencoder_1: REAL;
	
	(*the status word for GSTAT*)
	
	status_1:DWORD;
	status_2:DWORD;
	status_3:DWORD;
	status_4:DWORD;
	status_5:DWORD;
	status_6:DWORD;
	fb_diagnose_111: MB_ReadParameter;
	str_diagnose_11: DWORD;
	fb_blink_diagnos_11: BLINK;
	fb_diagnose_11: MB_ReadrealParameter;
	str_diagnose_111: REAL;
	fb_readpar_speed_2: MB_ReadRealParameter;
	fb_readpar_speed_4: MB_ReadRealParameter;
	fb_readpar_speed_6: MB_ReadRealParameter;
	
	ReadAxisPshape: ARRAY[1..5] OF MB_ReadlrealParameter;
	ReadAxisVact: ARRAY[1..5] OF MB_ReadlrealParameter;
	ReadAxisVshape: ARRAY[1..5] OF MB_ReadlrealParameter;

	conut_i: INT;
	b_PID_in_FI: BOOL;
	b_limit_cw_FI: BOOL;
	b_limit_ccw_FI: BOOL;
	b_limit_final_FI: BOOL;
	fb_readpar_pos_cmd_1: MB_ReadRealParameter;
END_VAR

P_GSTAT_K2STAT.A_Read_Parameter();

status_code1:=LEFT(str_diagnose_1,5);
status_code2:=LEFT(str_diagnose_2,5);
status_code3:=LEFT(str_diagnose_3,5);
status_code4:=LEFT(str_diagnose_4,5);
status_code5:=LEFT(str_diagnose_5,5);
status_code6:=LEFT(str_diagnose_6,5);

FOR  conut_i:=1 TO 5 BY 1 DO
ReadAxisPshape[conut_i](
	Enable:=axisdata[1].Axis_Inbb , 
	Done=> , 
	Active=> , 
	Error=> , 
	ErrorID=> , 
	ErrorIdent=> , 
	ParameterNumber:=FP_P_0_0434 , 
	Value=>P_shape_value[conut_i] , 
	Axis:=AxRef[conut_i] );
	
ReadAxisVshape[conut_i](
	Enable:=axisdata[1].Axis_Inbb , 
	Done=> , 
	Active=> , 
	Error=> , 
	ErrorID=> , 
	ErrorIdent=> , 
	ParameterNumber:=FP_P_0_0434 , 
	Value=>V_shape_value[conut_i] , 
	Axis:=AxRef[conut_i] );
	
ReadAxisVact[conut_i](
	Enable:=axisdata[1].Axis_Inbb , 
	Done=> , 
	Active=> , 
	Error=> , 
	ErrorID=> , 
	ErrorIdent=> , 
	ParameterNumber:=FP_S_0_0040 , 
	Value=>V_act_value[conut_i] , 
	Axis:=AxRef[conut_i] );
END_FOR

(*<<<<<<<<<<<<<<<<<<<<<<<<<<<<<master_status>>>>>>>>>>>>>>>>>>>>>>>>>>>>>>>>>>>>>>>>>>>>>>>>>>>>>>>*)
master_status.0:=axisdata[1].Axis_InAb;
IF b_remote_on=TRUE THEN
	master_status.1:=0;
ELSE
	master_status.1:=1;
END_IF
IF b_DSdoor_Estop  THEN
	master_status.2:=1;
ELSE
	master_status.2:=0;
END_IF

IF ABS(axisdata[3].rActualPosition_i-90)<0.02 THEN
	master_status.3:=1;
ELSE
	master_status.3:=0;
END_IF
	master_status.4:=(axisdata[1].Axis_Error OR axisdata[2].Axis_Error OR axisdata[3].Axis_Error OR axisdata[4].Axis_Error OR axisdata[5].Axis_Error OR axisdata[6].Axis_Error);
	master_status.5:=b_stow_pin_limit_unlock;
	master_status.6:=b_stow_pin_limit_lock;
	
IF i_num_stack_left>9500 THEN
		master_status.7:=0;
	ELSE IF i_num_stack_left<1500 THEN
		master_status.7:=1;	
	END_IF
		
END_IF

IF b_remote_on_run AND b_track_on THEN
	master_status.9:=0;
	master_status.8:=1;
ELSIF b_remote_on_run AND b_Track_Pause = TRUE THEN
	master_status.9:=1;
	master_status.8:=0;
ELSIF b_remote_on_run AND b_Track_Pause = FALSE  AND b_track_on = FALSE THEN
	master_status.9:=0;
	master_status.8:=0;
ELSE
 	master_status.9:=1;
	master_status.8:=1;
END_IF

IF 	b_encoder_ok_az	AND b_encoder_ok_FI THEN
	master_status.10:=1;
	master_status.11:=1;
ELSIF b_encoder_ok_az =FALSE AND b_encoder_ok_FI THEN
	master_status.10:=0;
	master_status.11:=1;
ELSIF b_encoder_ok_az  AND b_encoder_ok_FI=FALSE THEN
	master_status.10:=1;
	master_status.11:=0;
ELSE
	master_status.10:=0;
	master_status.11:=0;		
END_IF

IF b_remote_on_run THEN
	master_status.12:=1;
ELSE
	master_status.12:=0;
END_IF
	
IF b_remote_on_run THEN
	master_status.12:=1;
ELSE
	master_status.12:=0;
END_IF

IF b_permit_new_file THEN
	master_status.13:=1;
ELSE
	master_status.13:=0;
END_IF

(*<<<<<<<<<<<<<<<<<<<<<<<<<<<<<status_1>>>>>>>>>>>>>>>>>>>>>>>>>>>>>>>>>>>>>>>>>>>>>>>>>>>>>>>*)
status_1.0:=axisdata[1].Axis_InAb;
status_1.1:=b_PID_in_az;
status_1.2:=dw_brake_1.0;
status_1.3:=b_limit_cw_az;
status_1.4:=b_limit_ccw_az;
status_1.5:=(b_limit_final_cw_az OR b_limit_final_ccw_az);
status_1.6:=axisdata[1].Axis_Error;

(*<<<<<<<<<<<<<<<<<<<<<<<<<<<<<status_2>>>>>>>>>>>>>>>>>>>>>>>>>>>>>>>>>>>>>>>>>>>>>>>>>>>>>>>*)
status_2.0:=axisdata[2].Axis_InAb;
status_2.1:=b_PID_in_az;
status_2.2:=dw_brake_2.0;
status_2.3:=b_limit_cw_az;
status_2.4:=b_limit_ccw_az;
status_2.5:=(b_limit_final_cw_az OR b_limit_final_ccw_az);
status_2.6:=axisdata[2].Axis_Error;

(*<<<<<<<<<<<<<<<<<<<<<<<<<<<<<status_3>>>>>>>>>>>>>>>>>>>>>>>>>>>>>>>>>>>>>>>>>>>>>>>>>>>>>>>*)
status_3.0:=axisdata[3].Axis_InAb;
status_3.1:=b_PID_in_el;
status_3.2:=dw_brake_3.0;
status_3.3:=b_limit_cw_el;
status_3.4:=b_limit_ccw_el;
status_3.5:=(b_limit_final_cw_el OR b_limit_final_ccw_el) ;
status_3.6:=axisdata[3].Axis_Error;

(*<<<<<<<<<<<<<<<<<<<<<<<<<<<<<status_4>>>>>>>>>>>>>>>>>>>>>>>>>>>>>>>>>>>>>>>>>>>>>>>>>>>>>>>*)
status_4.0:=axisdata[4].Axis_InAb;
status_4.1:=b_PID_in_el;
status_4.2:=dw_brake_4.0;
status_4.3:=b_limit_cw_el;
status_4.4:=b_limit_ccw_el;
status_4.5:=(b_limit_final_cw_el OR b_limit_final_ccw_el); 
status_4.6:=axisdata[4].Axis_Error;

(*<<<<<<<<<<<<<<<<<<<<<<<<<<<<<status_5>>>>>>>>>>>>>>>>>>>>>>>>>>>>>>>>>>>>>>>>>>>>>>>>>>>>>>>*)
status_5.0:=axisdata[5].Axis_InAb;
status_5.1:=b_PID_in_FI;
status_5.2:=dw_brake_5.0;
status_5.3:=b_limit_cw_FI;
status_5.4:=b_limit_ccw_FI;
status_5.5:=b_limit_final_FI;
status_5.6:=axisdata[5].Axis_Error;

(*<<<<<<<<<<<<<<<<<<<<<<<<<<<<<status_6>>>>>>>>>>>>>>>>>>>>>>>>>>>>>>>>>>>>>>>>>>>>>>>>>>>>>>>*)
status_6.0:=axisdata[6].Axis_InAb;
status_6.1:=b_PID_in_FI;
status_6.2:=dw_brake_6.0;
status_6.3:=b_limit_cw_FI;
status_6.4:=b_limit_ccw_FI;
status_6.5:=b_limit_final_FI;
status_6.6:=axisdata[6].Axis_Error;


(*
(*<<<<<<<<<<<<<<<<<<<<<<<<<<<<<status_2>>>>>>>>>>>>>>>>>>>>>>>>>>>>>>>>>>>>>>>>>>>>>>>>>>>>>>>*)
status_2.0:=NOT(axisdata[2].Axis_InAb);
status_2.1:=axisdata[2].Axis_Error;
status_2.2:=NOT(dw_brake_2.0);
IF r_temp_motor2>120 THEN
status_2.3:=1;
b_power_Az:=FALSE;
b_enable_az_1:=FALSE;
b_enable_az_2:=FALSE;
ELSE
status_2.3:=0;
END_IF
IF r_current_2>5 THEN
status_2.4:=1;
ELSE
status_2.4:=0;
END_IF
(*<<<<<<<<<<<<<<<<<<<<<<<<<<<<<status_3>>>>>>>>>>>>>>>>>>>>>>>>>>>>>>>>>>>>>>>>>>>>>>>>>>>>>>>*)
status_3.0:=NOT(axisdata[3].Axis_InAb);
status_3.1:=axisdata[3].Axis_Error;
status_3.2:=NOT(dw_brake_3.0);
IF r_temp_motor3>120 THEN
status_3.3:=1;
b_power_El:=FALSE;
b_enable_el_3:=FALSE;
b_enable_el_4:=FALSE;
ELSE
status_3.3:=0;
END_IF
IF r_current_3>5 THEN
status_3.4:=1;
ELSE
status_3.4:=0;
END_IF
status_3.8:=NOT(b_PID_in_el);

IF (b_scc_goto=TRUE AND (b_goto_Az_done=FALSE OR b_goto_El_done=FALSE OR b_goto_FI_done=FALSE)) OR (b_track_on=TRUE AND i_num_stack_left<>0) THEN
status_3.9:=1;
END_IF;
IF (b_goto_Az_done=TRUE AND b_goto_El_done=TRUE AND b_goto_FI_done=TRUE) OR i_num_stack_left=0 THEN
status_3.9:=0;
END_IF;

status_3.10:=NOT(b_track_on);
IF ABS(r_track_error[2])<0.0034 THEN
	status_3.11:=0;
ELSE
	status_3.11:=1;
END_IF
status_3.12:=axisdata[3].Axis_Error;
IF ABS(r_following_3)>0.5 THEN
status_3.13:=1;
ELSE
status_3.13:=0;
END_IF
IF r_pos_el<14.6 THEN
	status_3.14:=1;
ELSE
	status_3.14:=0;
END_IF
IF r_pos_el>90.15 THEN
	status_3.15:=1;
ELSE
	status_3.15:=0;
END_IF
status_3.16:=b_limit_ccw_el;
status_3.17:=b_limit_cw_el;
status_3.18:=b_limit_final_el;
status_3.19:=b_track_overspeed_el;
(*<<<<<<<<<<<<<<<<<<<<<<<<<<<<<status_4>>>>>>>>>>>>>>>>>>>>>>>>>>>>>>>>>>>>>>>>>>>>>>>>>>>>>>>*)
status_4.0:=NOT(axisdata[4].Axis_InAb);
status_4.1:=axisdata[4].Axis_Error;
status_4.2:=NOT(dw_brake_4.0);
IF r_temp_motor4>120 THEN
status_4.3:=1;
b_power_El:=FALSE;
b_enable_el_3:=FALSE;
b_enable_el_4:=FALSE;
ELSE
status_4.3:=0;
END_IF
IF r_current_4>5 THEN
status_4.4:=1;
ELSE
status_4.4:=0;
END_IF
(*<<<<<<<<<<<<<<<<<<<<<<<<<<<<<status_5>>>>>>>>>>>>>>>>>>>>>>>>>>>>>>>>>>>>>>>>>>>>>>>>>>>>>>>*)
status_5.0:=NOT(axisdata[5].Axis_InAb);
status_5.1:=axisdata[5].Axis_Error;
status_5.2:=NOT(dw_brake_5.0);
IF r_temp_motor5>120 THEN
status_5.3:=1;
b_power_FI:=FALSE;
b_enable_FI_5:=FALSE;
ELSE
status_5.3:=0;
END_IF
IF r_current_5>5 THEN
status_5.4:=1;
ELSE
status_5.4:=0;
END_IF

status_5.8:=NOT(b_gearinpos_5_done);

IF (b_scc_goto=TRUE AND (b_goto_Az_done=FALSE OR b_goto_El_done=FALSE OR b_goto_FI_done=FALSE)) OR (b_track_on=TRUE AND i_num_stack_left<>0) THEN
status_5.9:=1;
END_IF;
IF (b_goto_Az_done=TRUE AND b_goto_El_done=TRUE AND b_goto_FI_done=TRUE) OR i_num_stack_left=0 THEN
status_5.9:=0;
END_IF;

status_5.10:=NOT(b_track_on);
IF ABS(r_track_error[3])<0.0034 THEN
	status_5.11:=0;
ELSE
	status_5.11:=1;
END_IF
status_5.12:=axisdata[5].Axis_Error;
IF ABS(r_following_5)>0.5 THEN
status_5.13:=1;
ELSE
status_5.13:=0;
END_IF

IF r_pos_FI<-89 THEN
	status_5.14:=1;
ELSE
	status_5.14:=0;
END_IF

IF r_pos_FI>89 THEN
	status_5.15:=1;
ELSE
	status_5.15:=0;
END_IF
status_5.16:=b_limit_ccw_FI;
status_5.17:=b_limit_cw_FI;
status_5.18:=b_limit_final_FI;
status_5.19:=b_track_overspeed_FI;
*)

(*<<<<<<<<<<<<<<<<<<<<<<<<<<<<<concatenate STR_GSTAT>>>>>>>>>>>>>>>>>>>>>>>>>>>>>>>>>>>>>>>>>>>>>>>>>>>>>>>*)
str_concat[1]:=CONCAT(' ',DWORD_TO_STRING(status_1));
str_concat[2]:=CONCAT(' ',LREAL_TO_STRING(F_reduce_to_1_bit(LREAL_TO_STRING(r_current_1))));
str_concat[3]:=CONCAT(' ',LREAL_TO_STRING(r_temp_motor1));
str_concat[4]:=CONCAT(' ',LREAL_TO_STRING(i_speed_1));
str_concat[5]:=CONCAT(' ',LREAL_TO_STRING(F_reduce_to_1_bit(LREAL_TO_STRING(r_motorencoder_1))));


str_concat[6]:=CONCAT(' ',DWORD_TO_STRING(status_2));
str_concat[7]:=CONCAT(' ',LREAL_TO_STRING(F_reduce_to_1_bit(LREAL_TO_STRING(r_current_2))));
str_concat[8]:=CONCAT(' ',LREAL_TO_STRING(r_temp_motor2));
str_concat[9]:=CONCAT(' ',LREAL_TO_STRING(i_speed_2));
str_concat[10]:=CONCAT(' ',LREAL_TO_STRING(F_reduce_to_1_bit(LREAL_TO_STRING(r_motorencoder_2))));

str_concat[11]:=CONCAT(' ',DWORD_TO_STRING(status_3));
str_concat[12]:=CONCAT(' ',LREAL_TO_STRING(F_reduce_to_1_bit(LREAL_TO_STRING(r_current_3))));
str_concat[13]:=CONCAT(' ',LREAL_TO_STRING(r_temp_motor3));
str_concat[14]:=CONCAT(' ',LREAL_TO_STRING(i_speed_3));
str_concat[15]:=CONCAT(' ',LREAL_TO_STRING(F_reduce_to_1_bit(LREAL_TO_STRING(r_motorencoder_3))));

str_concat[16]:=CONCAT(' ',DWORD_TO_STRING(status_4));
str_concat[17]:=CONCAT(' ',LREAL_TO_STRING(F_reduce_to_1_bit(LREAL_TO_STRING(r_current_4))));
str_concat[18]:=CONCAT(' ',LREAL_TO_STRING(r_temp_motor4));
str_concat[19]:=CONCAT(' ',LREAL_TO_STRING(i_speed_4));
str_concat[20]:=CONCAT(' ',LREAL_TO_STRING(F_reduce_to_1_bit(LREAL_TO_STRING(r_motorencoder_4))));

str_concat[21]:=CONCAT(' ',DWORD_TO_STRING(status_5));
str_concat[22]:=CONCAT(' ',LREAL_TO_STRING(F_reduce_to_1_bit(LREAL_TO_STRING(r_current_5))));
str_concat[23]:=CONCAT(' ',LREAL_TO_STRING(r_temp_motor5));
str_concat[24]:=CONCAT(' ',LREAL_TO_STRING(i_speed_5));
str_concat[25]:=CONCAT(' ',LREAL_TO_STRING(F_reduce_to_1_bit(LREAL_TO_STRING(r_motorencoder_5))));

str_concat[26]:=CONCAT(' ',DWORD_TO_STRING(status_6));
str_concat[27]:=CONCAT(' ',LREAL_TO_STRING(F_reduce_to_1_bit(LREAL_TO_STRING(r_current_6))));
str_concat[28]:=CONCAT(' ',LREAL_TO_STRING(r_temp_motor6));
str_concat[29]:=CONCAT(' ',LREAL_TO_STRING(i_speed_6));
str_concat[30]:=CONCAT(' ',LREAL_TO_STRING(F_reduce_to_1_bit(LREAL_TO_STRING(r_motorencoder_6))));

str_concat[31]:=CONCAT(' ',last_command);
str_concat[32]:=CONCAT(' ',INT_TO_STRING(i_receive_cmd));
str_concat[33]:=CONCAT(' ',INT_TO_STRING(i_excute_cmd));
(*
str_concat[31]:=CONCAT(' ',REAL_TO_STRING(F_reduce_to_4_bit(REAL_TO_STRING(r_test1))));
str_concat[32]:=CONCAT(' ',REAL_TO_STRING(F_reduce_to_4_bit(REAL_TO_STRING(r_test2))));
str_concat[33]:=CONCAT(' ',REAL_TO_STRING(F_reduce_to_4_bit(REAL_TO_STRING(r_test3))));
*)
STR_GSTAT_M:='';(*for语句格式*)
				FOR Counter:=1 TO 33 BY 1 DO
					STR_GSTAT_M:=CONCAT(STR_GSTAT_M,str_concat[Counter]);
				END_FOR;



(*
STR_GSTAT:=CONCAT(STR_GSTAT,CONCAT(' ',DWORD_TO_STRING(status_1)));
STR_GSTAT:=CONCAT(STR_GSTAT,CONCAT(' ',REAL_TO_STRING(r_current_1)));
STR_GSTAT:=CONCAT(STR_GSTAT,CONCAT(' ',REAL_TO_STRING(r_temp_motor1)));
STR_GSTAT:=CONCAT(STR_GSTAT,CONCAT(' ',REAL_TO_STRING(i_speed_1)));
*)


(*
STR_GSTAT:=CONCAT(STR_GSTAT,CONCAT(' ',DWORD_TO_STRING(status_2)));
STR_GSTAT:=CONCAT(STR_GSTAT,CONCAT(' ',REAL_TO_STRING(r_current_2)));
STR_GSTAT:=CONCAT(STR_GSTAT,CONCAT(' ',REAL_TO_STRING(r_temp_motor2)));
STR_GSTAT:=CONCAT(STR_GSTAT,CONCAT(' ',REAL_TO_STRING(i_speed_1)));

STR_GSTAT:=CONCAT(STR_GSTAT,CONCAT(' ',DWORD_TO_STRING(status_3)));
STR_GSTAT:=CONCAT(STR_GSTAT,CONCAT(' ',REAL_TO_STRING(r_current_3)));
STR_GSTAT:=CONCAT(STR_GSTAT,CONCAT(' ',REAL_TO_STRING(r_temp_motor3)));
STR_GSTAT:=CONCAT(STR_GSTAT,CONCAT(' ',REAL_TO_STRING(i_speed_3)));

STR_GSTAT:=CONCAT(STR_GSTAT,CONCAT(' ',DWORD_TO_STRING(status_4)));
STR_GSTAT:=CONCAT(STR_GSTAT,CONCAT(' ',REAL_TO_STRING(r_current_4)));
STR_GSTAT:=CONCAT(STR_GSTAT,CONCAT(' ',REAL_TO_STRING(r_temp_motor4)));
STR_GSTAT:=CONCAT(STR_GSTAT,CONCAT(' ',REAL_TO_STRING(i_speed_3)));

STR_GSTAT:=CONCAT(STR_GSTAT,CONCAT(' ',DWORD_TO_STRING(status_5)));
STR_GSTAT:=CONCAT(STR_GSTAT,CONCAT(' ',REAL_TO_STRING(r_current_5)));
STR_GSTAT:=CONCAT(STR_GSTAT,CONCAT(' ',REAL_TO_STRING(r_temp_motor5)));
STR_GSTAT:=CONCAT(STR_GSTAT,CONCAT(' ',REAL_TO_STRING(i_speed_5)));

STR_GSTAT:=CONCAT(STR_GSTAT,CONCAT(' ',DWORD_TO_STRING(status_6)));
STR_GSTAT:=CONCAT(STR_GSTAT,CONCAT(' ',REAL_TO_STRING(r_current_6)));
STR_GSTAT:=CONCAT(STR_GSTAT,CONCAT(' ',REAL_TO_STRING(r_temp_motor6)));
STR_GSTAT:=CONCAT(STR_GSTAT,CONCAT(' ',REAL_TO_STRING(i_speed_5)));

STR_GSTAT:=CONCAT(STR_GSTAT,CONCAT(' ',INT_TO_STRING(i_num_stack_left)));
STR_GSTAT:=CONCAT(STR_GSTAT,CONCAT(' ',INT_TO_STRING(i_start)));
STR_GSTAT_M:=CONCAT(STR_GSTAT,CONCAT(' ',INT_TO_STRING(i_end)));

*)
(*<<<<<<<<<<<<<<<<<<<<<<<<<<<<<concatenate STR_K2STAT>>>>>>>>>>>>>>>>>>>>>>>>>>>>>>>>>>>>>>>>>>>>>>>>>>>>>>>*)
STR_K2STAT:=CONCAT('OK - ',REAL_TO_STRING(r_operation_hour/100));
STR_K2STAT:=CONCAT(STR_K2STAT,CONCAT(' ',LREAL_TO_STRING(r_temp_motor1)));
STR_K2STAT:=CONCAT(STR_K2STAT,CONCAT(' ',LREAL_TO_STRING(r_temp_motor2)));
STR_K2STAT:=CONCAT(STR_K2STAT,CONCAT(' ',LREAL_TO_STRING(r_temp_motor3)));
STR_K2STAT:=CONCAT(STR_K2STAT,CONCAT(' ',LREAL_TO_STRING(r_temp_motor4)));
STR_K2STAT:=CONCAT(STR_K2STAT,CONCAT(' ',LREAL_TO_STRING(r_temp_motor5)));
STR_K2STAT:=CONCAT(STR_K2STAT,CONCAT(' ',LREAL_TO_STRING(r_temp_amp1)));
STR_K2STAT:=CONCAT(STR_K2STAT,CONCAT(' ',LREAL_TO_STRING(r_temp_amp2)));
STR_K2STAT:=CONCAT(STR_K2STAT,CONCAT(' ',LREAL_TO_STRING(r_temp_amp3)));
STR_K2STAT:=CONCAT(STR_K2STAT,CONCAT(' ',LREAL_TO_STRING(r_temp_amp4)));
STR_K2STAT:=CONCAT(STR_K2STAT,CONCAT(' ',LREAL_TO_STRING(r_temp_amp5)));
STR_K2STAT_M:=CONCAT(STR_K2STAT,CONCAT(' ',LREAL_TO_STRING(r_temp_MLC)));
(*<<<<<<<<<<<<<<<<<<<<<<<<<<<<<concatenate STR_K4STAT>>>>>>>>>>>>>>>>>>>>>>>>>>>>>>>>>>>>>>>>>>>>>>>>>>>>>>>*)
STR_K4STAT:=CONCAT('OK - ',str_diagnose_MLC);
STR_K4STAT:=CONCAT(STR_K4STAT,CONCAT(' ',str_diagnose_1));
STR_K4STAT:=CONCAT(STR_K4STAT,CONCAT(' ',str_diagnose_2));
STR_K4STAT:=CONCAT(STR_K4STAT,CONCAT(' ',str_diagnose_3));
STR_K4STAT:=CONCAT(STR_K4STAT,CONCAT(' ',str_diagnose_4));
STR_K4STAT_M:=CONCAT(STR_K4STAT,CONCAT(' ',str_diagnose_5));

(*<<<<<<<<<<<<<<<<<<<<<<<<<<<<<concatenate STR_K5STAT>>>>>>>>>>>>>>>>>>>>>>>>>>>>>>>>>>>>>>>>>>>>>>>>>>>>>>>*)
IF i_software_limit_1=16 AND i_hardware_limit_1=3 AND i_ESTOP_1=5 THEN
	b_azimuth_limit:=TRUE;
ELSE
	b_azimuth_limit:=FALSE;
END_IF

IF i_software_limit_3=16 AND i_hardware_limit_3=3 AND i_ESTOP_3=5 THEN
	b_elevation_limit:=TRUE;
ELSE
	b_elevation_limit:=FALSE;
END_IF

IF i_software_limit_5=16 AND i_hardware_limit_5=3 AND i_ESTOP_5=5 THEN
	b_FeedIndexer_limit:=TRUE;
ELSE
	b_FeedIndexer_limit:=FALSE;
END_IF
IF b_azimuth_limit AND b_elevation_limit AND b_FeedIndexer_limit THEN
	STR_K5STAT_M:='All the axes are safe.';
ELSE
	STR_K5STAT_M:='';
	IF b_azimuth_limit=FALSE THEN
		STR_K5STAT_M:=CONCAT(STR_K5STAT_M,'Azimuth axis is unsafe. ');
	END_IF
	IF b_elevation_limit=FALSE THEN
		STR_K5STAT_M:=CONCAT(STR_K5STAT_M,'Elevation axis is unsafe. ');
	END_IF
	IF b_FeedIndexer_limit=FALSE THEN
		STR_K5STAT_M:=CONCAT(STR_K5STAT_M,'FeedIndexer axis is unsafe. ');
	END_IF
END_IF

ACTION A_Read_Parameter:
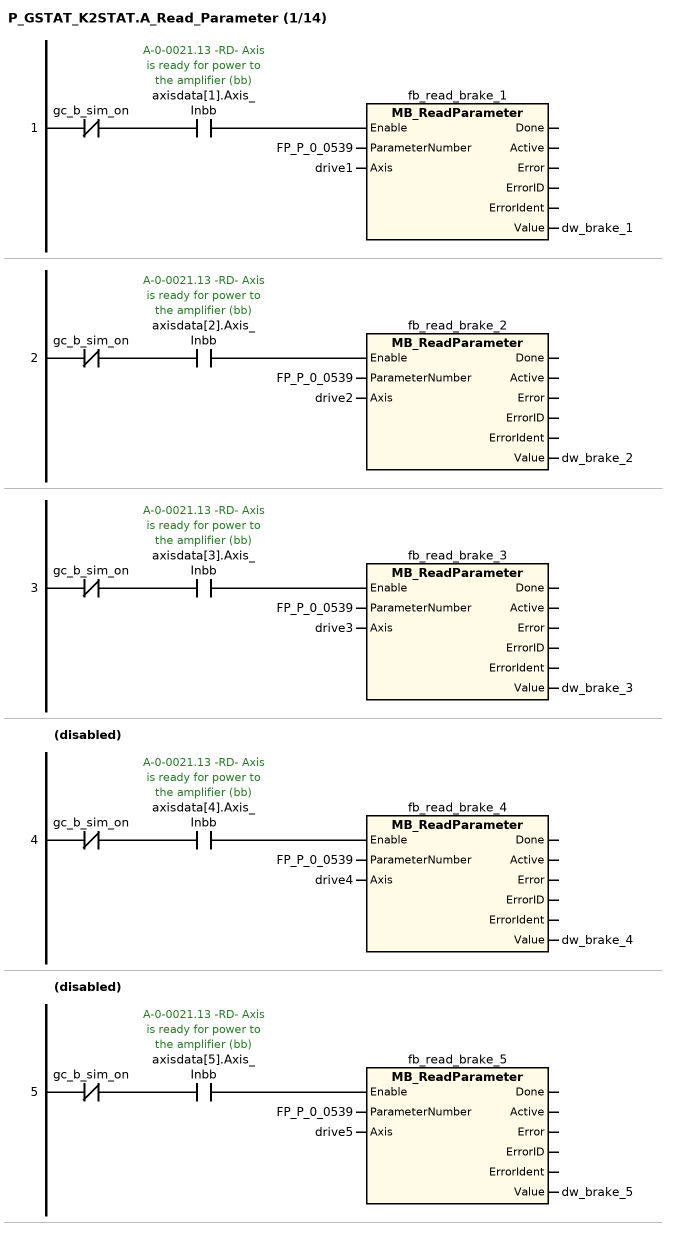
// NETWORK 1
//   fb_read_brake_1: With the function block "MB_ReadParameter" it is possible to read the current value of a parameter. The return value is DINT
//   axisdata[1].Axis_Inbb: A-0-0021.13 -RD- Axis is ready for power to the amplifier (bb)
//   FP_P_0_0539: Holding brake status word
//   drive1: Real axis "Drive1" with axis number 1
//   dw_brake_1: FP_P_0_0539,Holding brake status word
fb_read_brake_1(
    Enable := NOT gc_b_sim_on AND axisdata[1].Axis_Inbb,
    ParameterNumber := FP_P_0_0539,
    Axis := drive1,
    Value => dw_brake_1); // MB_ReadParameter

// NETWORK 2
//   axisdata[2].Axis_Inbb: A-0-0021.13 -RD- Axis is ready for power to the amplifier (bb)
//   FP_P_0_0539: Holding brake status word
//   drive2: Real axis "Drive2" with axis number 2
fb_read_brake_2(
    Enable := NOT gc_b_sim_on AND axisdata[2].Axis_Inbb,
    ParameterNumber := FP_P_0_0539,
    Axis := drive2,
    Value => dw_brake_2); // MB_ReadParameter

// NETWORK 3
//   axisdata[3].Axis_Inbb: A-0-0021.13 -RD- Axis is ready for power to the amplifier (bb)
//   FP_P_0_0539: Holding brake status word
//   drive3: Real axis "Drive3" with axis number 3
fb_read_brake_3(
    Enable := NOT gc_b_sim_on AND axisdata[3].Axis_Inbb,
    ParameterNumber := FP_P_0_0539,
    Axis := drive3,
    Value => dw_brake_3); // MB_ReadParameter

// NETWORK 4 (disabled)
//   axisdata[4].Axis_Inbb: A-0-0021.13 -RD- Axis is ready for power to the amplifier (bb)
//   FP_P_0_0539: Holding brake status word
//   drive4: Real axis "Drive4" with axis number 4
// fb_read_brake_4(
//     Enable := NOT gc_b_sim_on AND axisdata[4].Axis_Inbb,
//     ParameterNumber := FP_P_0_0539,
//     Axis := drive4,
//     Value => dw_brake_4); // MB_ReadParameter

// NETWORK 5 (disabled)
//   axisdata[5].Axis_Inbb: A-0-0021.13 -RD- Axis is ready for power to the amplifier (bb)
//   FP_P_0_0539: Holding brake status word
//   drive5: Real axis "Drive5" with axis number 5
// fb_read_brake_5(
//     Enable := NOT gc_b_sim_on AND axisdata[5].Axis_Inbb,
//     ParameterNumber := FP_P_0_0539,
//     Axis := drive5,
//     Value => dw_brake_5); // MB_ReadParameter

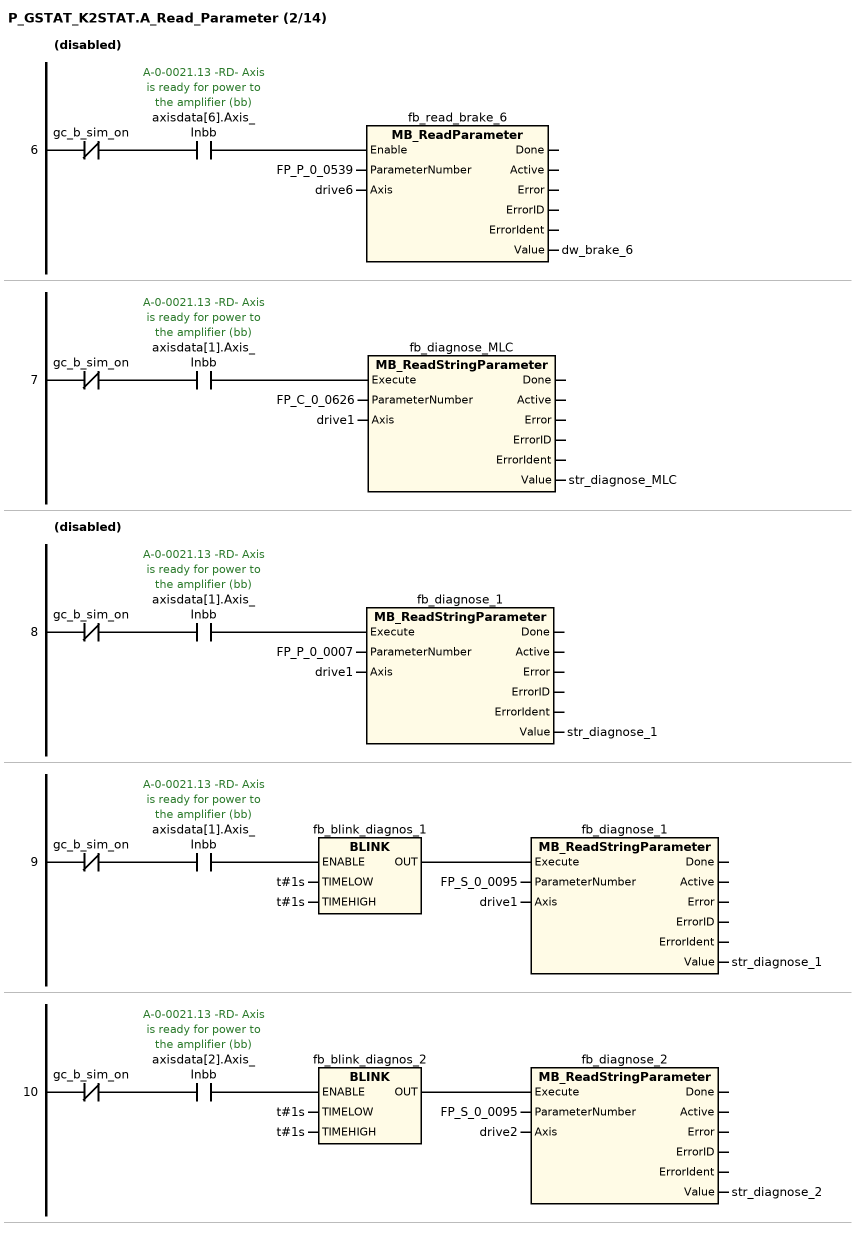
// NETWORK 6 (disabled)
//   axisdata[6].Axis_Inbb: A-0-0021.13 -RD- Axis is ready for power to the amplifier (bb)
//   FP_P_0_0539: Holding brake status word
//   drive6: Real axis "Drive6" with axis number 6
// fb_read_brake_6(
//     Enable := NOT gc_b_sim_on AND axisdata[6].Axis_Inbb,
//     ParameterNumber := FP_P_0_0539,
//     Axis := drive6,
//     Value => dw_brake_6); // MB_ReadParameter

// NETWORK 7
//   axisdata[1].Axis_Inbb: A-0-0021.13 -RD- Axis is ready for power to the amplifier (bb)
//   FP_C_0_0626: Diagnostics
//   drive1: Real axis "Drive1" with axis number 1
//   str_diagnose_MLC: FP_P_0_0007,Display text of diagnostic message
fb_diagnose_MLC(
    Execute := NOT gc_b_sim_on AND axisdata[1].Axis_Inbb,
    ParameterNumber := FP_C_0_0626,
    Axis := drive1,
    Value => str_diagnose_MLC); // MB_ReadStringParameter

// NETWORK 8 (disabled)
//   fb_diagnose_1: With the function block "MB_ReadStringParameter" it is possible to read a parameter the operating data of which has the ASCII format (string).
//   axisdata[1].Axis_Inbb: A-0-0021.13 -RD- Axis is ready for power to the amplifier (bb)
//   FP_P_0_0007: Display text of diagnostic message
//   drive1: Real axis "Drive1" with axis number 1
// fb_diagnose_1(
//     Execute := NOT gc_b_sim_on AND axisdata[1].Axis_Inbb,
//     ParameterNumber := FP_P_0_0007,
//     Axis := drive1,
//     Value => str_diagnose_1); // MB_ReadStringParameter

// NETWORK 9
//   fb_diagnose_1: With the function block "MB_ReadStringParameter" it is possible to read a parameter the operating data of which has the ASCII format (string).
//   fb_blink_diagnos_1: The function block BLINK generates a pulsating signal.The input consists of ENABLE of the type BOOL, as well as TIMELOW and TIMEHIGH of the type TIME.
//   axisdata[1].Axis_Inbb: A-0-0021.13 -RD- Axis is ready for power to the amplifier (bb)
//   FP_S_0_0095: Diagnostic message
//   drive1: Real axis "Drive1" with axis number 1
fb_blink_diagnos_1(ENABLE := NOT gc_b_sim_on AND axisdata[1].Axis_Inbb, TIMELOW := t#1s, TIMEHIGH := t#1s); // BLINK
fb_diagnose_1(
    Execute := fb_blink_diagnos_1.OUT,
    ParameterNumber := FP_S_0_0095,
    Axis := drive1,
    Value => str_diagnose_1); // MB_ReadStringParameter

// NETWORK 10
//   axisdata[2].Axis_Inbb: A-0-0021.13 -RD- Axis is ready for power to the amplifier (bb)
//   FP_S_0_0095: Diagnostic message
//   drive2: Real axis "Drive2" with axis number 2
fb_blink_diagnos_2(ENABLE := NOT gc_b_sim_on AND axisdata[2].Axis_Inbb, TIMELOW := t#1s, TIMEHIGH := t#1s); // BLINK
fb_diagnose_2(
    Execute := fb_blink_diagnos_2.OUT,
    ParameterNumber := FP_S_0_0095,
    Axis := drive2,
    Value => str_diagnose_2); // MB_ReadStringParameter

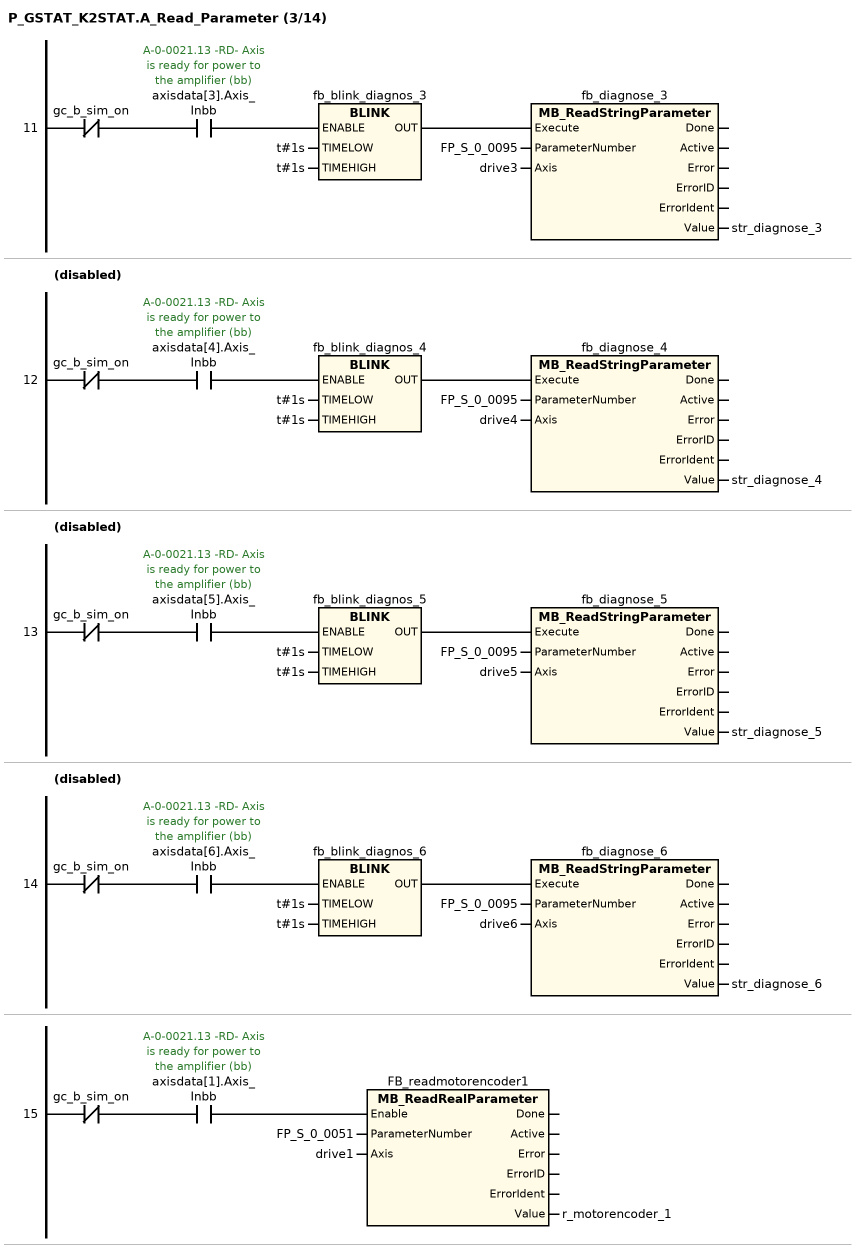
// NETWORK 11
//   axisdata[3].Axis_Inbb: A-0-0021.13 -RD- Axis is ready for power to the amplifier (bb)
//   FP_S_0_0095: Diagnostic message
//   drive3: Real axis "Drive3" with axis number 3
fb_blink_diagnos_3(ENABLE := NOT gc_b_sim_on AND axisdata[3].Axis_Inbb, TIMELOW := t#1s, TIMEHIGH := t#1s); // BLINK
fb_diagnose_3(
    Execute := fb_blink_diagnos_3.OUT,
    ParameterNumber := FP_S_0_0095,
    Axis := drive3,
    Value => str_diagnose_3); // MB_ReadStringParameter

// NETWORK 12 (disabled)
//   axisdata[4].Axis_Inbb: A-0-0021.13 -RD- Axis is ready for power to the amplifier (bb)
//   FP_S_0_0095: Diagnostic message
//   drive4: Real axis "Drive4" with axis number 4
// fb_blink_diagnos_4(ENABLE := NOT gc_b_sim_on AND axisdata[4].Axis_Inbb, TIMELOW := t#1s, TIMEHIGH := t#1s); // BLINK
// fb_diagnose_4(
//     Execute := fb_blink_diagnos_4.OUT,
//     ParameterNumber := FP_S_0_0095,
//     Axis := drive4,
//     Value => str_diagnose_4); // MB_ReadStringParameter

// NETWORK 13 (disabled)
//   axisdata[5].Axis_Inbb: A-0-0021.13 -RD- Axis is ready for power to the amplifier (bb)
//   FP_S_0_0095: Diagnostic message
//   drive5: Real axis "Drive5" with axis number 5
// fb_blink_diagnos_5(ENABLE := NOT gc_b_sim_on AND axisdata[5].Axis_Inbb, TIMELOW := t#1s, TIMEHIGH := t#1s); // BLINK
// fb_diagnose_5(
//     Execute := fb_blink_diagnos_5.OUT,
//     ParameterNumber := FP_S_0_0095,
//     Axis := drive5,
//     Value => str_diagnose_5); // MB_ReadStringParameter

// NETWORK 14 (disabled)
//   axisdata[6].Axis_Inbb: A-0-0021.13 -RD- Axis is ready for power to the amplifier (bb)
//   FP_S_0_0095: Diagnostic message
//   drive6: Real axis "Drive6" with axis number 6
// fb_blink_diagnos_6(ENABLE := NOT gc_b_sim_on AND axisdata[6].Axis_Inbb, TIMELOW := t#1s, TIMEHIGH := t#1s); // BLINK
// fb_diagnose_6(
//     Execute := fb_blink_diagnos_6.OUT,
//     ParameterNumber := FP_S_0_0095,
//     Axis := drive6,
//     Value => str_diagnose_6); // MB_ReadStringParameter

// NETWORK 15
//   axisdata[1].Axis_Inbb: A-0-0021.13 -RD- Axis is ready for power to the amplifier (bb)
//   FP_S_0_0051: Position feedback value 1
//   drive1: Real axis "Drive1" with axis number 1
FB_readmotorencoder1(
    Enable := NOT gc_b_sim_on AND axisdata[1].Axis_Inbb,
    ParameterNumber := FP_S_0_0051,
    Axis := drive1,
    Value => r_motorencoder_1); // MB_ReadRealParameter

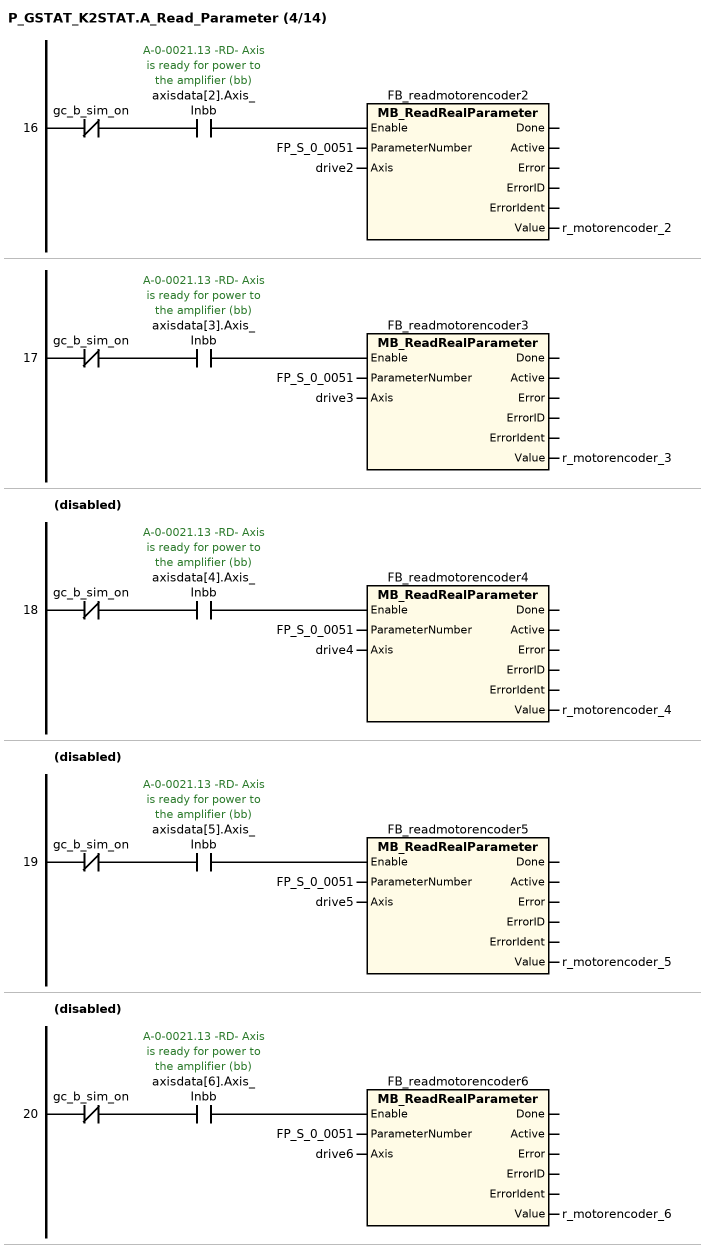
// NETWORK 16
//   axisdata[2].Axis_Inbb: A-0-0021.13 -RD- Axis is ready for power to the amplifier (bb)
//   FP_S_0_0051: Position feedback value 1
//   drive2: Real axis "Drive2" with axis number 2
FB_readmotorencoder2(
    Enable := NOT gc_b_sim_on AND axisdata[2].Axis_Inbb,
    ParameterNumber := FP_S_0_0051,
    Axis := drive2,
    Value => r_motorencoder_2); // MB_ReadRealParameter

// NETWORK 17
//   axisdata[3].Axis_Inbb: A-0-0021.13 -RD- Axis is ready for power to the amplifier (bb)
//   FP_S_0_0051: Position feedback value 1
//   drive3: Real axis "Drive3" with axis number 3
FB_readmotorencoder3(
    Enable := NOT gc_b_sim_on AND axisdata[3].Axis_Inbb,
    ParameterNumber := FP_S_0_0051,
    Axis := drive3,
    Value => r_motorencoder_3); // MB_ReadRealParameter

// NETWORK 18 (disabled)
//   axisdata[4].Axis_Inbb: A-0-0021.13 -RD- Axis is ready for power to the amplifier (bb)
//   FP_S_0_0051: Position feedback value 1
//   drive4: Real axis "Drive4" with axis number 4
// FB_readmotorencoder4(
//     Enable := NOT gc_b_sim_on AND axisdata[4].Axis_Inbb,
//     ParameterNumber := FP_S_0_0051,
//     Axis := drive4,
//     Value => r_motorencoder_4); // MB_ReadRealParameter

// NETWORK 19 (disabled)
//   axisdata[5].Axis_Inbb: A-0-0021.13 -RD- Axis is ready for power to the amplifier (bb)
//   FP_S_0_0051: Position feedback value 1
//   drive5: Real axis "Drive5" with axis number 5
// FB_readmotorencoder5(
//     Enable := NOT gc_b_sim_on AND axisdata[5].Axis_Inbb,
//     ParameterNumber := FP_S_0_0051,
//     Axis := drive5,
//     Value => r_motorencoder_5); // MB_ReadRealParameter

// NETWORK 20 (disabled)
//   axisdata[6].Axis_Inbb: A-0-0021.13 -RD- Axis is ready for power to the amplifier (bb)
//   FP_S_0_0051: Position feedback value 1
//   drive6: Real axis "Drive6" with axis number 6
// FB_readmotorencoder6(
//     Enable := NOT gc_b_sim_on AND axisdata[6].Axis_Inbb,
//     ParameterNumber := FP_S_0_0051,
//     Axis := drive6,
//     Value => r_motorencoder_6); // MB_ReadRealParameter

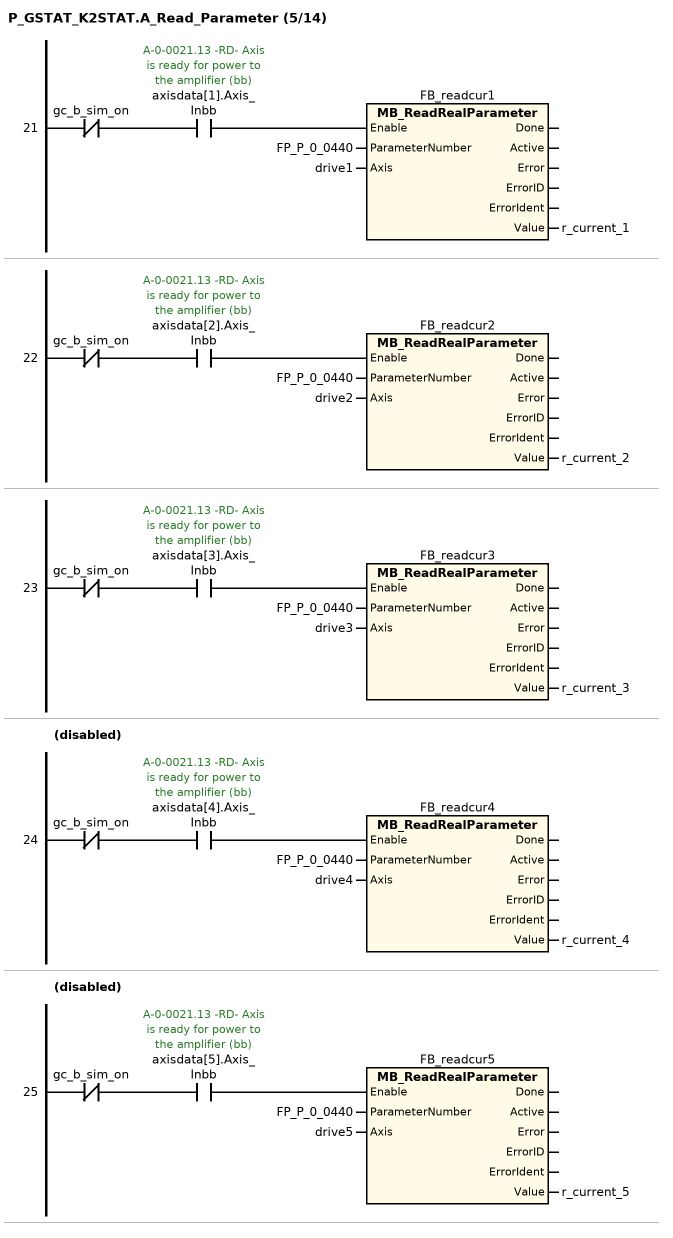
// NETWORK 21
//   FB_readcur1: With the function block "MB_ReadRealParameter" it is possible to read the current value of a parameter. The return value is REAL.
//   axisdata[1].Axis_Inbb: A-0-0021.13 -RD- Axis is ready for power to the amplifier (bb)
//   FP_P_0_0440: Actual output current value (absolute value)
//   drive1: Real axis "Drive1" with axis number 1
//   r_current_1: FP_P_0_0440,Actual output current value absolute value
FB_readcur1(
    Enable := NOT gc_b_sim_on AND axisdata[1].Axis_Inbb,
    ParameterNumber := FP_P_0_0440,
    Axis := drive1,
    Value => r_current_1); // MB_ReadRealParameter

// NETWORK 22
//   axisdata[2].Axis_Inbb: A-0-0021.13 -RD- Axis is ready for power to the amplifier (bb)
//   FP_P_0_0440: Actual output current value (absolute value)
//   drive2: Real axis "Drive2" with axis number 2
FB_readcur2(
    Enable := NOT gc_b_sim_on AND axisdata[2].Axis_Inbb,
    ParameterNumber := FP_P_0_0440,
    Axis := drive2,
    Value => r_current_2); // MB_ReadRealParameter

// NETWORK 23
//   axisdata[3].Axis_Inbb: A-0-0021.13 -RD- Axis is ready for power to the amplifier (bb)
//   FP_P_0_0440: Actual output current value (absolute value)
//   drive3: Real axis "Drive3" with axis number 3
FB_readcur3(
    Enable := NOT gc_b_sim_on AND axisdata[3].Axis_Inbb,
    ParameterNumber := FP_P_0_0440,
    Axis := drive3,
    Value => r_current_3); // MB_ReadRealParameter

// NETWORK 24 (disabled)
//   axisdata[4].Axis_Inbb: A-0-0021.13 -RD- Axis is ready for power to the amplifier (bb)
//   FP_P_0_0440: Actual output current value (absolute value)
//   drive4: Real axis "Drive4" with axis number 4
// FB_readcur4(
//     Enable := NOT gc_b_sim_on AND axisdata[4].Axis_Inbb,
//     ParameterNumber := FP_P_0_0440,
//     Axis := drive4,
//     Value => r_current_4); // MB_ReadRealParameter

// NETWORK 25 (disabled)
//   axisdata[5].Axis_Inbb: A-0-0021.13 -RD- Axis is ready for power to the amplifier (bb)
//   FP_P_0_0440: Actual output current value (absolute value)
//   drive5: Real axis "Drive5" with axis number 5
// FB_readcur5(
//     Enable := NOT gc_b_sim_on AND axisdata[5].Axis_Inbb,
//     ParameterNumber := FP_P_0_0440,
//     Axis := drive5,
//     Value => r_current_5); // MB_ReadRealParameter

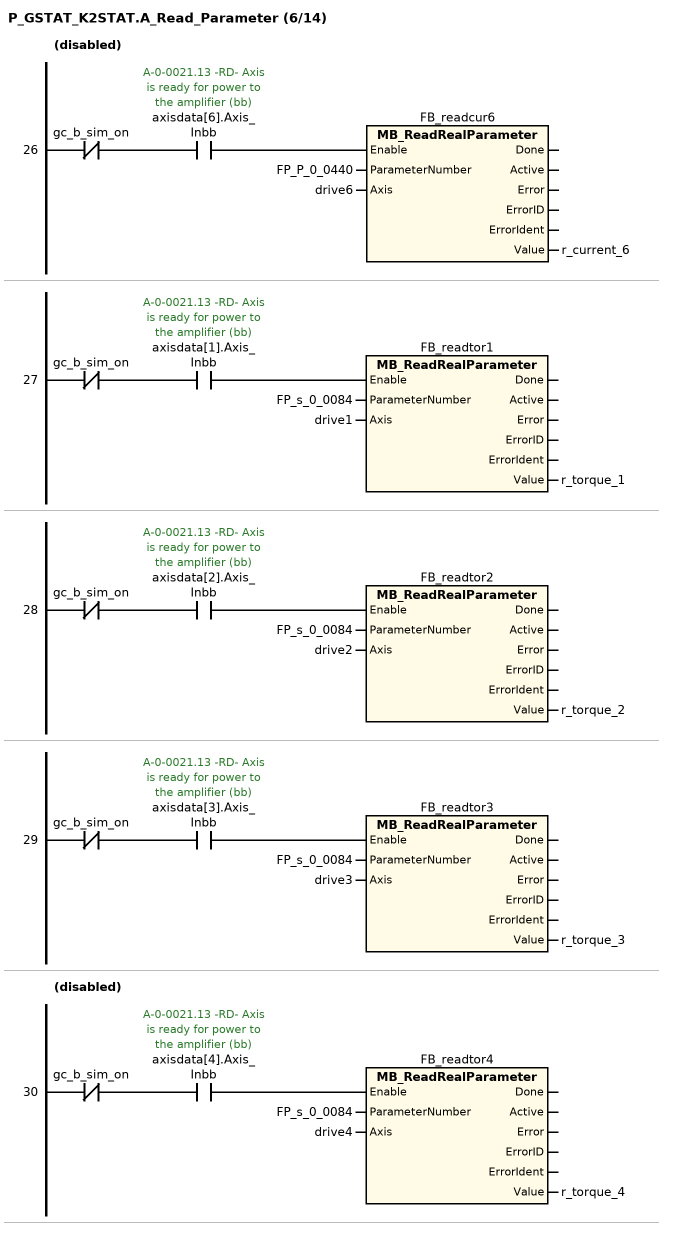
// NETWORK 26 (disabled)
//   axisdata[6].Axis_Inbb: A-0-0021.13 -RD- Axis is ready for power to the amplifier (bb)
//   FP_P_0_0440: Actual output current value (absolute value)
//   drive6: Real axis "Drive6" with axis number 6
// FB_readcur6(
//     Enable := NOT gc_b_sim_on AND axisdata[6].Axis_Inbb,
//     ParameterNumber := FP_P_0_0440,
//     Axis := drive6,
//     Value => r_current_6); // MB_ReadRealParameter

// NETWORK 27
//   axisdata[1].Axis_Inbb: A-0-0021.13 -RD- Axis is ready for power to the amplifier (bb)
//   FP_s_0_0084: Torque/force feedback value
//   drive1: Real axis "Drive1" with axis number 1
//   r_torque_1: FP_S_0_0084,Torque force feedback value
FB_readtor1(
    Enable := NOT gc_b_sim_on AND axisdata[1].Axis_Inbb,
    ParameterNumber := FP_s_0_0084,
    Axis := drive1,
    Value => r_torque_1); // MB_ReadRealParameter

// NETWORK 28
//   axisdata[2].Axis_Inbb: A-0-0021.13 -RD- Axis is ready for power to the amplifier (bb)
//   FP_s_0_0084: Torque/force feedback value
//   drive2: Real axis "Drive2" with axis number 2
FB_readtor2(
    Enable := NOT gc_b_sim_on AND axisdata[2].Axis_Inbb,
    ParameterNumber := FP_s_0_0084,
    Axis := drive2,
    Value => r_torque_2); // MB_ReadRealParameter

// NETWORK 29
//   axisdata[3].Axis_Inbb: A-0-0021.13 -RD- Axis is ready for power to the amplifier (bb)
//   FP_s_0_0084: Torque/force feedback value
//   drive3: Real axis "Drive3" with axis number 3
FB_readtor3(
    Enable := NOT gc_b_sim_on AND axisdata[3].Axis_Inbb,
    ParameterNumber := FP_s_0_0084,
    Axis := drive3,
    Value => r_torque_3); // MB_ReadRealParameter

// NETWORK 30 (disabled)
//   axisdata[4].Axis_Inbb: A-0-0021.13 -RD- Axis is ready for power to the amplifier (bb)
//   FP_s_0_0084: Torque/force feedback value
//   drive4: Real axis "Drive4" with axis number 4
// FB_readtor4(
//     Enable := NOT gc_b_sim_on AND axisdata[4].Axis_Inbb,
//     ParameterNumber := FP_s_0_0084,
//     Axis := drive4,
//     Value => r_torque_4); // MB_ReadRealParameter

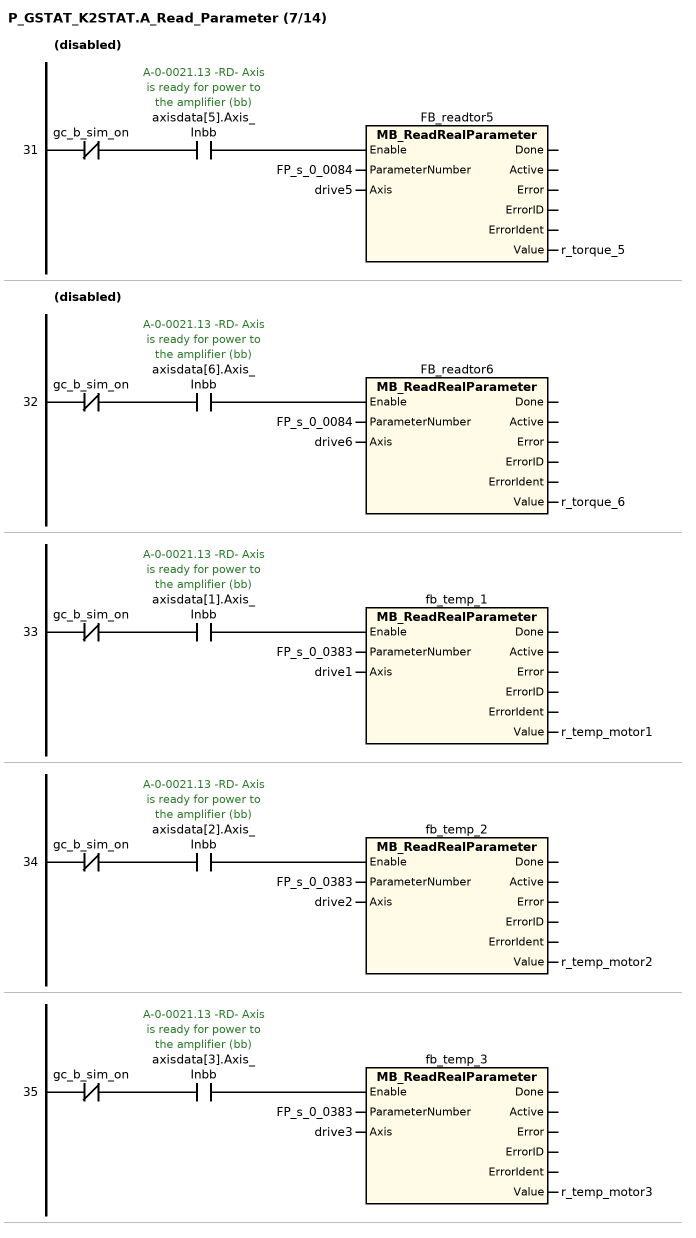
// NETWORK 31 (disabled)
//   axisdata[5].Axis_Inbb: A-0-0021.13 -RD- Axis is ready for power to the amplifier (bb)
//   FP_s_0_0084: Torque/force feedback value
//   drive5: Real axis "Drive5" with axis number 5
// FB_readtor5(
//     Enable := NOT gc_b_sim_on AND axisdata[5].Axis_Inbb,
//     ParameterNumber := FP_s_0_0084,
//     Axis := drive5,
//     Value => r_torque_5); // MB_ReadRealParameter

// NETWORK 32 (disabled)
//   axisdata[6].Axis_Inbb: A-0-0021.13 -RD- Axis is ready for power to the amplifier (bb)
//   FP_s_0_0084: Torque/force feedback value
//   drive6: Real axis "Drive6" with axis number 6
// FB_readtor6(
//     Enable := NOT gc_b_sim_on AND axisdata[6].Axis_Inbb,
//     ParameterNumber := FP_s_0_0084,
//     Axis := drive6,
//     Value => r_torque_6); // MB_ReadRealParameter

// NETWORK 33
//   axisdata[1].Axis_Inbb: A-0-0021.13 -RD- Axis is ready for power to the amplifier (bb)
//   FP_s_0_0383: Motor temperature
//   drive1: Real axis "Drive1" with axis number 1
//   r_temp_motor1: FP_S_0_0383,Motor temperature
fb_temp_1(
    Enable := NOT gc_b_sim_on AND axisdata[1].Axis_Inbb,
    ParameterNumber := FP_s_0_0383,
    Axis := drive1,
    Value => r_temp_motor1); // MB_ReadRealParameter

// NETWORK 34
//   axisdata[2].Axis_Inbb: A-0-0021.13 -RD- Axis is ready for power to the amplifier (bb)
//   FP_s_0_0383: Motor temperature
//   drive2: Real axis "Drive2" with axis number 2
fb_temp_2(
    Enable := NOT gc_b_sim_on AND axisdata[2].Axis_Inbb,
    ParameterNumber := FP_s_0_0383,
    Axis := drive2,
    Value => r_temp_motor2); // MB_ReadRealParameter

// NETWORK 35
//   axisdata[3].Axis_Inbb: A-0-0021.13 -RD- Axis is ready for power to the amplifier (bb)
//   FP_s_0_0383: Motor temperature
//   drive3: Real axis "Drive3" with axis number 3
fb_temp_3(
    Enable := NOT gc_b_sim_on AND axisdata[3].Axis_Inbb,
    ParameterNumber := FP_s_0_0383,
    Axis := drive3,
    Value => r_temp_motor3); // MB_ReadRealParameter

